            "8" : Bool;
            "9" : Bool;
            "10" : Bool;
            "11" : Bool;
            "12" : Bool;
            "13" : Bool;
            "14" : Bool;
            "15" : Bool;
            "16" : Bool;
         END_STRUCT;
         Spare_4 : Struct
            "1" : Bool;
            "2" : Bool;
            "3" : Bool;
            "4" : Bool;
            "5" : Bool;
            "6" : Bool;
            "7" : Bool;
            "8" : Bool;
            "9" : Bool;
            "10" : Bool;
            "11" : Bool;
            "12" : Bool;
            "13" : Bool;
            "14" : Bool;
            "15" : Bool;
            "16" : Bool;
         END_STRUCT;
      END_STRUCT;
      MES_Error : Struct
         Offline : Bool;   // MES离线
         Reserved1_8 : Bool;
         CheckInCompOverTime_1 : Bool;   // 心跳故障
         CheckInResultOverTime_1 : Bool;
         CheckInCompOverTime_2 : Bool;   // 二维码对比失败
         CheckInResultOverTime_2 : Bool;   // 获取打标数据NG
         CheckInCompOverTime_3 : Bool;   // 获取打标数据超时
         CheckInResultOverTime_3 : Bool;   // 缓存数据和MES数据对比不合格，步序错误 需初始化
         CheckInCompOverTime_4 : Bool;
         CheckInResultOverTime_4 : Bool;   // 主件查询完成超时
         CheckInCompOverTime_5 : Bool;   // 主件查询结果NG
         CheckInResultOverTime_5 : Bool;   // 主件查询完成复位超时
         CheckInCompOverTime_6 : Bool;
         CheckInResultOverTime_6 : Bool;
         CheckInCompOverTime_7 : Bool;
         CheckInResultOverTime_7 : Bool;   // 主件保存完成超时
         CheckInCompOverTime_8 : Bool;   // 主件保存结果反馈超时
         CheckInResultOverTime_8 : Bool;   // 主件保存触发错误
         CheckoutSaveResultNG : Bool;   // 主件保存结果NG
         CheckoutCompRstOverTime : Bool;   // 主件保存完成复位超时
         Reserved2_5 : Bool;
         Reserved2_6 : Bool;
         Reserved2_7 : Bool;
         SubCheck_CompOverTime : Bool;   // 子件查询完成超时
         SubCheck_ResultOverTime : Bool;   // 子件查询结果反馈超时
         SubCheck_TriggerError : Bool;   // 子件查询触发错误
         SubCheck_CheckResultNG : Bool;   // 子件查询结果NG
         SubCheck_CompRstOverTime : Bool;   // 子件查询完成复位超时
         Reserved3_5 : Bool;
         Reserved3_6 : Bool;
         Reserved3_7 : Bool;
         Processing_CompOverTime : Bool;   // 加工不可逆标记完成超时
         Reserved4_1 : Bool;
         Processing_TriggerError : Bool;   // 加工不可逆标记触发错误
         Reserved4_3 : Bool;
         Processing_CompRstOverTime : Bool;   // 加工不可逆标记完成复位超时
         Reserved4_5 : Bool;
         Reserved4_6 : Bool;
         Reserved4_7 : Bool;
         Reserved5_0 : Bool;
         Reserved5_1 : Bool;
         Reserved5_2 : Bool;
         Reserved5_3 : Bool;
         Reserved5_4 : Bool;
         Reserved5_5 : Bool;
         Reserved5_6 : Bool;
         Reserved5_7 : Bool;
      END_STRUCT;
   END_VAR
BEGIN
END_DATA_BLOCK

DATA_BLOCK "ST10_GlobalError"   // DB1066
{ S7_Optimized_Access := 'FALSE' }
// stored: AutoNumber false
   VAR RETAIN
      COM : Struct
         MainPneumaticPressure1NOK : Bool;   // Main Pneumatic pressure 1 NOK,pls check inptut Ix.x,then check if the main valve is opened
         MainPneumaticPressure2NOK : Bool;   // Main Pneumatic pressure 2 NOK,pls check inptut Ix.x,then check if the main valve is opened
         MainPneumaticPressure3NOK : Bool;   // Main Pneumatic pressure 3 NOK,pls check inptut Ix.x,then check if the main valve is opened
         StationNotInHP : Bool;   // Station not in Home position,can't start cycle,pls check the Home positiong state
         CabinetTemperatureNotOk : Bool;   // Cabinet Temperature not OK, please check input Ix.x,then check if the cooling and fan is working
         CoolingUnitNotOk : Bool;   // Cooling unit not OK,pls check input Ix.x,then check if the cooling and fan is working
         RotateTablePositionNOK : Bool;   // The position of the rotate table is not correct after change mode.pls reset position by manual
         RotateTableNotInPosition : Bool;   // No position signal after rotate table Stopped,please check table position and input Ix.x
         StationHardwareError : Bool;
         ChangeStyleError : Bool;
         Reserve3 : Bool;
         Reserve4 : Bool;
         Reserve5 : Bool;
         Reserve6 : Bool;
         Reserve7 : Bool;
         Reserve8 : Bool;
         Reserve : Array[1..4, 0..15] of Bool;
      END_STRUCT;
      Hardware : Struct
         PNSlaveStation01 : Array[1..10] of Struct
            Error : Bool;   // PLC Local Module Error,please check the error module,PLC hardware configuration and online monitor the PLC error message
            Reserve1 : Bool;
            Reserve2 : Bool;
         END_STRUCT;
         COMM : Array[1..5] of Struct   // Communication
            CommunicationError : Bool;   // Serial Communication error,please check power, hardware configuration and connection cable
            NoReceive : Bool;   // Serial Communication receive no information, please check the module settings and communication equipment is the same, check the communication line is the intersection or straight line
            ReceiveWrong : Bool;   // Serial Communication receive the information is wrong, please check the data area is updated in real time
            Reserve1 : Bool;
            Reserve2 : Bool;
         END_STRUCT;
         PNSlaveStation02 : Array[1..10] of Struct   // Substation
            Error : Bool;   // SubStation Missing, please check power, hardware configuration and connection cable
            Reserve1 : Bool;   // SubStation error, please check Slave error code, check the error information in the PLC online hardware
            Reserve2 : Bool;
            Reserve3 : Bool;
         END_STRUCT;
         PNSlaveStation03 : Array[1..10] of Struct   // Remote I/O Error (远程I/O错误）
            Error : Bool;   // Remote I/O communication error, please check the power and communication cable, check the hardware configuration of PLC
            Reserve1 : Bool;   // Remote I/O error, please online monitor the PLC error message
            Reserve2 : Bool;
            Reserve3 : Bool;
         END_STRUCT;
         ValveIsland : Array[1..5] of Struct   // Valve Island Error（阀岛错误）
            SystemError : Bool;   // Valve island error, pls check the error code , check the error information in the PLC online hardware
            OffLine : Bool;   // Valve island is lost, pls check the island's cable , check valve island in PLC configuration and the actual agreement
            Reserve1 : Bool;
            Reserve2 : Bool;
         END_STRUCT;
      END_STRUCT;
      Safety : Struct
         "Robot 1 Estop" : Bool;   // Safety circuit not OK,pls check input Ix.x,then check if the safety circuit control on
         "Robot 2 Estop" : Bool;   // E-stop safety circuit not OK, please check input Ix.x, then reset safety circurt
         HMIEstopPBActivated : Bool;   // HMI Estop PB Activated，pls check input Ix.x,then check Estop button,if Estop button is close,pls open the Estop button
         TableEstopPB1Activated : Bool;   // HTable Estop PB1 Activated，pls check input Ix.x,then check Estop button,if Estop button is close,pls open the Estop button
         TableEstopPB2Activated : Bool;   // Table Estop PB2 Activated，pls check input Ix.x,then check Estop button,if Estop button is close,pls open the Estop button
         TableEstopPB3Activated : Bool;   // Table Estop PB3 Activated，pls check input Ix.x,then check Estop button,if Estop button is close,pls open the Estop button
         TableEstopPB4Activated : Bool;   // Table Estop PB4 Activated，pls check input Ix.x,then check Estop button,if Estop button is close,pls open the Estop button
         TableEstopPB5Activated : Bool;   // Table Estop PB5 Activated，pls check input Ix.x,then check Estop button,if Estop button is close,pls open the Estop button
         TableEstopPB6Activated : Bool;   // Table Estop PB6 Activated，pls check input Ix.x,then check Estop button,if Estop button is close,pls open the Estop button
         EStopSafety : Bool;
         TableEstopPB7Activated : Bool;
         TableEstopPB8Activated : Bool;
         TableEstopPB9Activated : Bool;
         StoveEstopActivated : Bool;
         "Robot 3 Estop" : Bool;
         Reserve9 : Bool;
         Reserve : Array[1..4, 0..15] of Bool;
      END_STRUCT;
      SafetyDoor : Struct
         "Type" : Array[1..5] of Struct   // Safety Door circuit type
            NotOk : Bool;   // Safety Door type [*] circuit not OK, please check input Ix.x, then reset safety circurt
            OpenInRunning : Bool;   // The safety door is opened when device Running,pls power on than initialize device
            Reserve1 : Bool;
            Reserve2 : Bool;
         END_STRUCT;
         No : Array[1..9] of Struct   // SafetyDoorNumber
            NotLock : Bool;   // Safety door lock is not lock，pls check input Ix.x，then check safety door lock output Qx.x
            Notlocked : Bool;   // Safety door lock is not unlock，pls check input Ix.x，then check safety door lock output Qx.x
            NotClose : Bool;   // Safety door is not close,pls check satety door lock position
            Reserve1 : Bool;
            Reserve2 : Bool;
         END_STRUCT;
         MaterialDoor : Struct
            NotLock_1 : Bool;
            NotClose_1 : Bool;
            NotLock_2 : Bool;
            NotClose_2 : Bool;
            NotLock_3 : Bool;
            NotClose_3 : Bool;
            NotLock_4 : Bool;
            NotClose_4 : Bool;
            NotLock_5 : Bool;
            NotClose_5 : Bool;
            NotLock_6 : Bool;
            NotClose_6 : Bool;
            NotLock_7 : Bool;
            NotClose_7 : Bool;
            NotLock_8 : Bool;
            NotClose_8 : Bool;
         END_STRUCT;
      END_STRUCT;
      LightCurtain : Array[1..5] of Struct
         ActivatedInRunning : Bool;   // Light curtain is Activated when device Running, pls power on than initialize device
         ActivatedInRotTableRun : Bool;   // Light curtain is Activated when rotate table running,please press the reset button to rotate the rotate table to position
         Error : Bool;   // Light curtain error,pls check the light curtain connection or check the error code
         Reserve1 : Bool;
         Reserve2 : Bool;
      END_STRUCT;
      Product : Array[1..5] of Struct
         TypeSelectionError : Bool;   // Product Type selection error,pls select the proper type
         TypeWrong : Bool;   // Product is not match current model, please make sure the product model is entered correctly
         NotforStation : Bool;   // Product not for this station,pls check if the Product is proper
         TypeAutoChangeError : Bool;
         Reserve2 : Bool;
      END_STRUCT;
      Fixture : Array[1..10] of Struct
         PositionError : Bool;   // Fixture [*] position error,pls put the fixture on proper positon
         TypeError : Bool;   // Fixture [*] tpye error,pls put the correct fixture into the tooling
         Reserve1 : Bool;
         Reserve2 : Bool;
      END_STRUCT;
      Breaker : Struct   // Power Breaker
         Trip : Array[1..16] of Bool;   // Breaker tripped, please check input Ix.x
      END_STRUCT;
   END_VAR
BEGIN
END_DATA_BLOCK

DATA_BLOCK "ST10_WarningDB"   // DB1068
{ S7_Optimized_Access := 'FALSE' }
// stored: AutoNumber false
   VAR RETAIN
      Global : Struct   // Global Warning（通用警告）
         "1" : Struct
            PartLack1 : Bool;   // The main part1 lack
            PartLack2 : Bool;   // The part2 lack
            PartLack3 : Bool;   // The part3 lack
            PartLack4 : Bool;   // The part4 lack
            PartLack5 : Bool;   // The part5 lack
            PartLack6 : Bool;   // The part6 lack
            PartLack7 : Bool;   // The part7 lack
            PartLack8 : Bool;   // The part8 lack
         END_STRUCT;
         "2" : Array[0..15] of Bool;
         "3" : Struct
            PartNoProperPosition1 : Bool;   // The main part1 no proper position
            PartNoProperPosition2 : Bool;   // The part2 no proper position
            PartNoProperPosition3 : Bool;   // The part3 no proper position
            PartNoProperPosition4 : Bool;   // The part4 no proper position
            PartNoProperPosition5 : Bool;   // The part5 no proper position
            PartNoProperPosition6 : Bool;   // The part6 no proper position
            PartNoProperPosition7 : Bool;   // The part7 no proper position
            PartNoProperPosition8 : Bool;   // The part8 no proper position
         END_STRUCT;
         "4" : Array[0..15] of Bool;
         "5" : Struct
            ChangoverDataInvalide : Bool;   // The changover data invalide
            PartDateInvalide : Bool;   // The part date invalide
            StationInHPToStart : Bool;   // The station has to be at base pos to start
            lastStationPartNok : Bool;   // The last station part is Nok
         END_STRUCT;
         "6" : Array[0..15] of Bool;
         "7" : Array[0..15] of Bool;
         "8" : Array[0..15] of Bool;
         "9" : Array[0..15] of Bool;
         "10" : Array[0..15] of Bool;
      END_STRUCT;
      IndexTable : Array[1..2, 0..15] of Bool;   // Indextable Warning（转台警告）
      Serve : Array[1..2, 0..15] of Bool;   // Serve Warning（伺服警告）
      Servepress : Array[1..2, 0..15] of Bool;   // Serve press Warning（伺服压机警告）
      "3AxisServoInterpolation" : Array[1..2, 0..15] of Bool;   // Servo Motor Risk Money(3 axis)Warning （伺服电机3轴差补系统警告）
      LaserWelding : Array[1..2, 0..15] of Bool;   // Laser Welding Warning(激光焊接机警告)
      LaserMarking : Array[1..2, 0..15] of Bool;   // Laser Marking Warning(激光打标机警告)
      Printer : Array[1..2, 0..15] of Bool;   // Printer Warning(打印机警告)
      Marking : Array[1..2, 0..15] of Bool;   // Marking Warning(标识机警告)
      Labelling : Array[1..2, 0..15] of Bool;   // Labelling Warning（贴标机警告）
      Dispensing : Array[1..2, 0..15] of Bool;   // Dispensing Warning（点胶警告）
      GreasingSystem : Array[1..2, 0..15] of Bool;   // Greasing System Warning(注油系统警告）
      HotWindSystem : Array[1..2, 0..15] of Bool;   // Hot Wind System Warning(热风系统警告）
      HighFrequencyHeating : Array[1..2, 0..15] of Bool;   // High Frequency Heating Warning（高频加热警告）
      Degaussing : Array[1..2, 0..15] of Bool;   // Degaussing Warning（消磁警告）
      BowlFeeder : Array[1..2, 0..15] of Bool;   // Bowl Feeder Warning（振动盘警告）
      Riveter : Array[1..2, 0..15] of Bool;   // Riveter Warning（铆接机警告）
      HydraulicSystem : Array[1..2, 0..15] of Bool;   // Hydraulic System Warning（液压系统警告）
      Robot : Array[1..2, 0..15] of Bool;   // Robot Warning（机器人警告）
      Camera : Array[1..2, 0..15] of Bool;   // Camera Warning(影像警告)
      Scannner : Array[1..2, 0..15] of Bool;   // Scannner Warning(读码警告)
      MeasureSensor : Array[1..2, 0..15] of Bool;   // Measure Sensor Warning(测量传感器警告)
      Leakage : Array[1..2, 0..15] of Bool;   // Leakage Warning（泄露测试仪警告）
      TestPowerSupply : Array[1..2, 0..15] of Bool;   // Test Power Supply Warning (测试电源警告）
      HighVoltageTester : Array[1..2, 0..15] of Bool;   // High Voltage Test Warning(高压测试警告）
      EOLfinalInspection : Array[1..2, 0..15] of Bool;   // EOL final inspection Warning（EOL终检测试警告）
      Screw : Array[1..2, 0..15] of Bool;   // Screw Warning(电动螺丝刀警告)
      "3AxisScrewEncoder" : Array[1..2, 0..15] of Bool;   // Screw Encoder(3 axis)Warning(螺丝刀编码器警告）
      Heating : Array[1..2, 0..15] of Bool;   // Heating Warning（加热警告）
      PressurizedOilAirCylinder : Array[1..2, 0..15] of Bool;   // Pressurized Oil-Air Cylinder Warning(气液增力缸警告）
      Moby : Array[1..2, 0..15] of Bool;   // Moby Warning(Moby警告)
      IPC : Array[1..2, 0..15] of Bool;   // IPC Warning（服务器警告）
      ValveIsland : Array[1..2, 0..15] of Bool;   // Valve island Warning (阀岛警告）
      RFID : Array[1..2, 0..15] of Bool;   // RFID Warning（无线射频识别警告）
      RemoteIO : Array[1..2, 0..15] of Bool;   // Remote I/O Warning（远程I/O警告）
      DPSlaveStation : Array[1..2, 0..15] of Bool;   // DP Slave Station Warning（DP从站警告）
      MSCOMM : Array[1..2, 0..15] of Bool;   // MSCOMM Warning（串口通讯警告）
      Flowtester : Array[1..2, 0..15] of Bool;   // Flow tester Warning（流量测试仪错误）
      CurrentsTester : Array[1..2, 0..15] of Bool;   // Currents Tester Warning(电流测试仪)）
      VoltageTester : Array[1..2, 0..15] of Bool;   // Voltage Tester Warning(电压测试仪)
      InductanceTester : Array[1..2, 0..15] of Bool;   // Inductance Tester Warning(电感测试仪)
      ResistanceTester : Array[1..2, 0..15] of Bool;   // Resistance Tester Warning(电阻测试仪)
      LCRTester : Array[1..2, 0..15] of Bool;   // LCR Test Warning(LCR测试)
      PressureDisplacementMonitor : Array[1..2, 0..15] of Bool;   // Pressure Displacement Monitor Warning(压力位移监控仪)
      UltrasonicWelding : Array[1..2, 0..15] of Bool;   // Ultrasonic Welding Warning(超声波焊接)
      ElectricResistanceWelding : Array[1..2, 0..15] of Bool;   // Electric Resistance Welding Warning(电阻焊)
   END_VAR
BEGIN
END_DATA_BLOCK

DATA_BLOCK "ST10_TipDB"   // DB1069
{ S7_Optimized_Access := 'FALSE' }
// stored: AutoNumber false
   VAR RETAIN
      Global : Struct
         "1" : Struct
            ControlOn : Bool;   // 7000:提示：设备未上电，请先按复位按钮，再按控制开按钮
            closesafetyDoor : Bool;   // 7001:提示：设备存在故障，请查看报警信息，消除故障，然后按复位按钮
            LockSafetyDoor : Bool;   // 7003:提示：设备未选择自动，请选择自动模式
            SelectAutoMode : Bool;   // 7005:提示：设备未启动，请启动自动运行
            SelectManualMode : Bool;
            AutoModeRunning : Bool;
            SafetyDoorLocked : Bool;
            SaferyDoorNotLocked : Bool;
            GoWP : Bool;
            Reset : Bool;
         END_STRUCT;
         "2" : Array[0..15] of Bool;
         "3" : Array[0..15] of Bool;
         "4" : Array[0..15] of Bool;
         "5" : Struct
            FuncrionDeactive1 : Bool;
            FuncrionDeactive2 : Bool;
            FuncrionDeactive3 : Bool;
            FuncrionDeactive4 : Bool;
            FuncrionDeactive5 : Bool;
            FuncrionDeactive6 : Bool;
            FuncrionDeactive7 : Bool;
            FuncrionDeactive8 : Bool;
         END_STRUCT;
         "6" : Array[0..15] of Bool;
         "7" : Struct
            ScanMainPartDMC1 : Bool;
            ScanPartDMC2 : Bool;
            ScanPartDMC3 : Bool;
            ScanPartDMC4 : Bool;
            ScanPartDMC5 : Bool;
            ScanPartDMC6 : Bool;
            ScanPartDMC7 : Bool;
            ScanPartDMC8 : Bool;
         END_STRUCT;
         "8" : Array[0..15] of Bool;
         "9" : Array[0..15] of Bool;
         "10" : Array[0..15] of Bool;
      END_STRUCT;
      OP1 : Struct   // ST70_B_提示信息
         "Take off product" : Bool;   // 请取下托盘上产品
         "Put product" : Bool;   // 请放入转向器壳体总成
         "Please scan the code" : Bool;   // 请扫转向器壳体总成二维码
         "Please apply Oil" : Bool;   // 请手持涂油工装涂油
         "Please take the O-ring" : Bool;   // 请取O型圈并安装完成
         "Please put in the powertrain" : Bool;   // 请扫转向器总成二维码
         Static_2 : Bool;
         "Please pre-screw" : Bool;   // 请安装转向器动力总成并预拧螺丝
         Static_1 : Bool;
         Static_3 : Bool;
         "Please press the button_1" : Bool;   // 请按下ST70-B启动按钮
         Reset : Bool;   // RFID状态数据未清除，请复位清除数据
      END_STRUCT;
      OP2 : Struct   // ST70_C_提示信息
         Static_4 : Bool;
         Static_2 : Bool;
         Static_3 : Bool;
         "Please press the button" : Bool;   // 请按下ST70_C启动按钮
         "Please press the trigger" : Bool;   // 请按下螺丝枪扳机拧紧螺丝
         "Please take the paint pen" : Bool;   // 请取出油漆笔划上标识
         "Please put back the paint pen" : Bool;   // 请划上标识后放回油漆笔
         Static_1 : Bool;
         "Please remove the product" : Bool;   // 产品报废,请取下产品
         "Please press the screw gun trigger" : Bool;   // 重新拧紧,请按下螺丝枪扳机
      END_STRUCT;
   END_VAR
BEGIN
   // Global."2"[0] : 7002:提示：未选择配方，请在换型页面选择配方
   // Global."2"[1] : 7004:提示：设备未初始化，请启动初始化
END_DATA_BLOCK

DATA_BLOCK "Parameter"   // DB170
{ S7_Optimized_Access := 'TRUE' }
// stored: AutoNumber false, IsRetainMemResEnabled true, MemoryReserve 10000
   VAR RETAIN
      AxisRun : Struct
         Axis : Array[1..15] of "ServoType_UDT";
      END_STRUCT;
      AxisNuw : Struct
         Axis : Array[1..15] of "ServoType_UDT";
      END_STRUCT;
      AxisDisplay : Struct
         Axis : Array[1..15] of "ServoType_UDT";
      END_STRUCT;
      AxisSave : Struct
         Axis : Array[1..15] of "ServoType_UDT";
      END_STRUCT;
      AxisStore : Array[1..15] of Struct
         Axis : Array[1..15] of "ServoType_UDT";
      END_STRUCT;
   END_VAR
BEGIN
   // AxisRun.Axis[1].Pos1 : 上料位1
   // AxisRun.Axis[2].Pos1 : 初始位
   // AxisRun.Axis[3].Pos1 : 初始位/IV拍照位_1
   // AxisRun.Axis[4].Pos1 : 上料位1
   // AxisRun.Axis[5].Pos1 : Z轴初始位
   // AxisRun.Axis[6].Pos1 : X轴初始位
   // AxisRun.Axis[7].Pos1 : Y轴初始位
   AxisRun.Axis[1].Pos1.Position := 3.419;
   AxisRun.Axis[2..3].Pos1.Position := 0.0;
   AxisRun.Axis[4].Pos1.Position := 3.585;
   AxisRun.Axis[5].Pos1.Position := 143.76;
   AxisRun.Axis[6].Pos1.Position := 2.34;
   AxisRun.Axis[7].Pos1.Position := 115.47;
   AxisRun.Axis[8..15].Pos1.Position := 0.0;
   AxisRun.Axis[1..2].Pos1.Speed := 10000;
   AxisRun.Axis[3].Pos1.Speed := 20000;
   AxisRun.Axis[4].Pos1.Speed := 10000;
   AxisRun.Axis[5..7].Pos1.Speed := 200;
   AxisRun.Axis[8..15].Pos1.Speed := 0;
   AxisRun.Axis[1..15].Pos1.Reached := FALSE;
   // AxisRun.Axis[1].Pos2 : 上料位2
   // AxisRun.Axis[2].Pos2 : 扫码位置2
   // AxisRun.Axis[3].Pos2 : 点胶1结束位
   // AxisRun.Axis[4].Pos2 : 上料位2
   // AxisRun.Axis[5].Pos2 : Z轴点胶位1
   // AxisRun.Axis[6].Pos2 : X轴点胶等待位
   // AxisRun.Axis[7].Pos2 : Y轴点胶位1
   AxisRun.Axis[1].Pos2.Position := 48.386;
   AxisRun.Axis[2].Pos2.Position := 450.0;
   AxisRun.Axis[3].Pos2.Position := 490.0;
   AxisRun.Axis[4].Pos2.Position := 48.61;
   AxisRun.Axis[5].Pos2.Position := 143.76;
   AxisRun.Axis[6].Pos2.Position := 76.0;
   AxisRun.Axis[7].Pos2.Position := 115.47;
   AxisRun.Axis[8..15].Pos2.Position := 0.0;
   AxisRun.Axis[1..4].Pos2.Speed := 10000;
   AxisRun.Axis[5..7].Pos2.Speed := 200;
   AxisRun.Axis[8..15].Pos2.Speed := 0;
   AxisRun.Axis[1..15].Pos2.Reached := FALSE;
   // AxisRun.Axis[1].Pos3 : 上料位3
   // AxisRun.Axis[2].Pos3 : 扫码位置3
   // AxisRun.Axis[3].Pos3 : 点胶2结束位
   // AxisRun.Axis[4].Pos3 : 上料位3
   // AxisRun.Axis[5].Pos3 : Z轴点胶位2
   // AxisRun.Axis[6].Pos3 : X轴点胶位1
   // AxisRun.Axis[7].Pos3 : Y轴点胶位2
   AxisRun.Axis[1].Pos3.Position := 93.294;
   AxisRun.Axis[2].Pos3.Position := 900.0;
   AxisRun.Axis[3].Pos3.Position := 490.0;
   AxisRun.Axis[4].Pos3.Position := 93.637;
   AxisRun.Axis[5].Pos3.Position := 137.76;
   AxisRun.Axis[6].Pos3.Position := 84.69;
   AxisRun.Axis[7].Pos3.Position := 115.47;
   AxisRun.Axis[8..15].Pos3.Position := 0.0;
   AxisRun.Axis[1..4].Pos3.Speed := 10000;
   AxisRun.Axis[5..7].Pos3.Speed := 200;
   AxisRun.Axis[8..15].Pos3.Speed := 0;
   AxisRun.Axis[1..15].Pos3.Reached := FALSE;
   // AxisRun.Axis[1].Pos4 : 上料位4
   // AxisRun.Axis[2].Pos4 : 扫码位置4
   // AxisRun.Axis[3].Pos4 : 点胶3结束位
   // AxisRun.Axis[4].Pos4 : 上料位4
   // AxisRun.Axis[5].Pos4 : Z轴点胶位3
   // AxisRun.Axis[6].Pos4 : X轴点胶位2
   // AxisRun.Axis[7].Pos4 : Y轴点胶位3
   AxisRun.Axis[1].Pos4.Position := 138.335;
   AxisRun.Axis[2].Pos4.Position := 135.0;
   AxisRun.Axis[3].Pos4.Position := 490.0;
   AxisRun.Axis[4].Pos4.Position := 138.606;
   AxisRun.Axis[5].Pos4.Position := 130.36;
   AxisRun.Axis[6].Pos4.Position := 84.69;
   AxisRun.Axis[7].Pos4.Position := 115.47;
   AxisRun.Axis[8..15].Pos4.Position := 0.0;
   AxisRun.Axis[1..4].Pos4.Speed := 10000;
   AxisRun.Axis[5..7].Pos4.Speed := 200;
   AxisRun.Axis[8..15].Pos4.Speed := 0;
   AxisRun.Axis[1..15].Pos4.Reached := FALSE;
   // AxisRun.Axis[1].Pos5 : 上料位5
   // AxisRun.Axis[2].Pos5 : 扫码位置5
   // AxisRun.Axis[3].Pos5 : 点胶4结束位//点胶位置取消
   // AxisRun.Axis[4].Pos5 : 上料位5
   // AxisRun.Axis[5].Pos5 : Z轴点胶位4
   // AxisRun.Axis[6].Pos5 : X轴点胶位3
   // AxisRun.Axis[7].Pos5 : Y轴点胶位4
   AxisRun.Axis[1].Pos5.Position := 183.464;
   AxisRun.Axis[2].Pos5.Position := 180.0;
   AxisRun.Axis[3].Pos5.Position := 0.0;
   AxisRun.Axis[4].Pos5.Position := 183.388;
   AxisRun.Axis[5].Pos5.Position := 124.16;
   AxisRun.Axis[6].Pos5.Position := 84.69;
   AxisRun.Axis[7].Pos5.Position := 115.47;
   AxisRun.Axis[8..15].Pos5.Position := 0.0;
   AxisRun.Axis[1..2].Pos5.Speed := 10000;
   AxisRun.Axis[3].Pos5.Speed := 0;
   AxisRun.Axis[4].Pos5.Speed := 10000;
   AxisRun.Axis[5..7].Pos5.Speed := 200;
   AxisRun.Axis[8..15].Pos5.Speed := 0;
   AxisRun.Axis[1..15].Pos5.Reached := FALSE;
   // AxisRun.Axis[1].Pos6 : 上料位6
   // AxisRun.Axis[2].Pos6 : 扫码位置6
   // AxisRun.Axis[3].Pos6 : 点胶5结束位
   // AxisRun.Axis[4].Pos6 : 上料位6
   // AxisRun.Axis[5].Pos6 : Z轴点胶位5
   // AxisRun.Axis[6].Pos6 : X轴点胶位4
   // AxisRun.Axis[7].Pos6 : Y轴点胶位5
   AxisRun.Axis[1].Pos6.Position := 228.443;
   AxisRun.Axis[2].Pos6.Position := 225.0;
   AxisRun.Axis[3].Pos6.Position := 490.0;
   AxisRun.Axis[4].Pos6.Position := 228.458;
   AxisRun.Axis[5].Pos6.Position := 125.65;
   AxisRun.Axis[6].Pos6.Position := 84.69;
   AxisRun.Axis[7].Pos6.Position := 110.18;
   AxisRun.Axis[8..15].Pos6.Position := 0.0;
   AxisRun.Axis[1..4].Pos6.Speed := 10000;
   AxisRun.Axis[5..7].Pos6.Speed := 200;
   AxisRun.Axis[8..15].Pos6.Speed := 0;
   AxisRun.Axis[1..15].Pos6.Reached := FALSE;
   // AxisRun.Axis[1].Pos7 : 上料位7
   // AxisRun.Axis[2].Pos7 : 扫码位置7
   // AxisRun.Axis[3].Pos7 : IV拍照位_2
   // AxisRun.Axis[4].Pos7 : 上料位7
   // AxisRun.Axis[5].Pos7 : Z轴相机检测位
   // AxisRun.Axis[6].Pos7 : X轴点胶位5
   // AxisRun.Axis[7].Pos7 : Y轴相机检测位
   AxisRun.Axis[1].Pos7.Position := 273.535;
   AxisRun.Axis[2].Pos7.Position := 270.0;
   AxisRun.Axis[3].Pos7.Position := 90.0;
   AxisRun.Axis[4].Pos7.Position := 273.513;
   AxisRun.Axis[5].Pos7.Position := 48.11;
   AxisRun.Axis[6].Pos7.Position := 85.0;
   AxisRun.Axis[7].Pos7.Position := 60.52;
   AxisRun.Axis[8..15].Pos7.Position := 0.0;
   AxisRun.Axis[1..4].Pos7.Speed := 10000;
   AxisRun.Axis[5..7].Pos7.Speed := 200;
   AxisRun.Axis[8..15].Pos7.Speed := 0;
   AxisRun.Axis[1..15].Pos7.Reached := FALSE;
   // AxisRun.Axis[1].Pos8 : 上料位8
   // AxisRun.Axis[2].Pos8 : 扫码位置8
   // AxisRun.Axis[3].Pos8 : IV拍照位_3
   // AxisRun.Axis[4].Pos8 : 上料位8
   // AxisRun.Axis[5].Pos8 : Z轴原点位
   // AxisRun.Axis[6].Pos8 : X轴相机检测位
   AxisRun.Axis[1].Pos8.Position := 318.25;
   AxisRun.Axis[2].Pos8.Position := 315.0;
   AxisRun.Axis[3].Pos8.Position := 180.0;
   AxisRun.Axis[4].Pos8.Position := 318.501;
   AxisRun.Axis[5].Pos8.Position := 0.0;
   AxisRun.Axis[6].Pos8.Position := 88.53;
   AxisRun.Axis[7].Pos8.Position := 80.0;
   AxisRun.Axis[8..15].Pos8.Position := 0.0;
   AxisRun.Axis[1..4].Pos8.Speed := 10000;
   AxisRun.Axis[5..6].Pos8.Speed := 200;
   AxisRun.Axis[7].Pos8.Speed := 100;
   AxisRun.Axis[8..15].Pos8.Speed := 0;
   AxisRun.Axis[1..15].Pos8.Reached := FALSE;
   // AxisRun.Axis[3].Pos9 : IV拍照位_4
   // AxisRun.Axis[5].Pos9 : Z轴Up点胶位5
   AxisRun.Axis[1..2].Pos9.Position := 0.0;
   AxisRun.Axis[3].Pos9.Position := 270.0;
   AxisRun.Axis[4].Pos9.Position := 0.0;
   AxisRun.Axis[5].Pos9.Position := 48.11;
   AxisRun.Axis[6..15].Pos9.Position := 0.0;
   AxisRun.Axis[1..2].Pos9.Speed := 0;
   AxisRun.Axis[3].Pos9.Speed := 10000;
   AxisRun.Axis[4].Pos9.Speed := 0;
   AxisRun.Axis[5].Pos9.Speed := 200;
   AxisRun.Axis[6..15].Pos9.Speed := 0;
   AxisRun.Axis[1..15].Pos9.Reached := FALSE;
   AxisRun.Axis[1..15].Pos10.Position := 0.0;
   AxisRun.Axis[1..15].Pos10.Speed := 0;
   AxisRun.Axis[1..15].Pos10.Reached := FALSE;
   AxisRun.Axis[1..15].Pos11.Position := 0.0;
   AxisRun.Axis[1..15].Pos11.Speed := 0;
   AxisRun.Axis[1..15].Pos11.Reached := FALSE;
   AxisRun.Axis[1..15].Pos12.Position := 0.0;
   AxisRun.Axis[1..15].Pos12.Speed := 0;
   AxisRun.Axis[1..15].Pos12.Reached := FALSE;
   AxisRun.Axis[1..15].Pos13.Position := 0.0;
   AxisRun.Axis[1..15].Pos13.Speed := 0;
   AxisRun.Axis[1..15].Pos13.Reached := FALSE;
   AxisRun.Axis[1..15].Pos14.Position := 0.0;
   AxisRun.Axis[1..15].Pos14.Speed := 0;
   AxisRun.Axis[1..15].Pos14.Reached := FALSE;
   AxisRun.Axis[1..15].Pos15.Position := 0.0;
   AxisRun.Axis[1..15].Pos15.Speed := 0;
   AxisRun.Axis[1..15].Pos15.Reached := FALSE;
   AxisRun.Axis[1..15].Pos16.Position := 0.0;
   AxisRun.Axis[1..15].Pos16.Speed := 0;
   AxisRun.Axis[1..15].Pos16.Reached := FALSE;
   AxisRun.Axis[1..15].Pos17.Position := 0.0;
   AxisRun.Axis[1..15].Pos17.Speed := 0;
   AxisRun.Axis[1..15].Pos17.Reached := FALSE;
   AxisRun.Axis[1..15].Pos18.Position := 0.0;
   AxisRun.Axis[1..15].Pos18.Speed := 0;
   AxisRun.Axis[1..15].Pos18.Reached := FALSE;
   AxisRun.Axis[1..15].Pos19.Position := 0.0;
   AxisRun.Axis[1..15].Pos19.Speed := 0;
   AxisRun.Axis[1..15].Pos19.Reached := FALSE;
   AxisRun.Axis[1..15].Pos20.Position := 0.0;
   AxisRun.Axis[1..15].Pos20.Speed := 0;
   AxisRun.Axis[1..15].Pos20.Reached := FALSE;
   AxisRun.Axis[1..15].Pos21.Position := 0.0;
   AxisRun.Axis[1..15].Pos21.Speed := 0;
   AxisRun.Axis[1..15].Pos21.Reached := FALSE;
   AxisRun.Axis[1..15].Pos22.Position := 0.0;
   AxisRun.Axis[1..15].Pos22.Speed := 0;
   AxisRun.Axis[1..15].Pos22.Reached := FALSE;
   AxisRun.Axis[1..15].Pos23.Position := 0.0;
   AxisRun.Axis[1..15].Pos23.Speed := 0;
   AxisRun.Axis[1..15].Pos23.Reached := FALSE;
   AxisRun.Axis[1..15].Pos24.Position := 0.0;
   AxisRun.Axis[1..15].Pos24.Speed := 0;
   AxisRun.Axis[1..15].Pos24.Reached := FALSE;
   AxisRun.Axis[1..15].Pos25.Position := 0.0;
   AxisRun.Axis[1..15].Pos25.Speed := 0;
   AxisRun.Axis[1..15].Pos25.Reached := FALSE;
   AxisRun.Axis[1..15].Pos26.Position := 0.0;
   AxisRun.Axis[1..15].Pos26.Speed := 0;
   AxisRun.Axis[1..15].Pos26.Reached := FALSE;
   AxisRun.Axis[1..15].Pos27.Position := 0.0;
   AxisRun.Axis[1..15].Pos27.Speed := 0;
   AxisRun.Axis[1..15].Pos27.Reached := FALSE;
   AxisRun.Axis[1..15].Pos28.Position := 0.0;
   AxisRun.Axis[1..15].Pos28.Speed := 0;
   AxisRun.Axis[1..15].Pos28.Reached := FALSE;
   AxisRun.Axis[1..15].Pos29.Position := 0.0;
   AxisRun.Axis[1..15].Pos29.Speed := 0;
   AxisRun.Axis[1..15].Pos29.Reached := FALSE;
   AxisRun.Axis[1..15].Pos30.Position := 0.0;
   AxisRun.Axis[1..15].Pos30.Speed := 0;
   AxisRun.Axis[1..15].Pos30.Reached := FALSE;
   AxisNuw.Axis[1..15].Pos1.Position := 0.0;
   AxisNuw.Axis[1..15].Pos1.Speed := 0;
   AxisNuw.Axis[1..15].Pos1.Reached := FALSE;
   AxisNuw.Axis[1..15].Pos2.Position := 0.0;
   AxisNuw.Axis[1..15].Pos2.Speed := 0;
   AxisNuw.Axis[1..15].Pos2.Reached := FALSE;
   AxisNuw.Axis[1..15].Pos3.Position := 0.0;
   AxisNuw.Axis[1..15].Pos3.Speed := 0;
   AxisNuw.Axis[1..15].Pos3.Reached := FALSE;
   AxisNuw.Axis[1..15].Pos4.Position := 0.0;
   AxisNuw.Axis[1..15].Pos4.Speed := 0;
   AxisNuw.Axis[1..15].Pos4.Reached := FALSE;
   AxisNuw.Axis[1..15].Pos5.Position := 0.0;
   AxisNuw.Axis[1..15].Pos5.Speed := 0;
   AxisNuw.Axis[1..15].Pos5.Reached := FALSE;
   AxisNuw.Axis[1..15].Pos6.Position := 0.0;
   AxisNuw.Axis[1..15].Pos6.Speed := 0;
   AxisNuw.Axis[1..15].Pos6.Reached := FALSE;
   AxisNuw.Axis[1..15].Pos7.Position := 0.0;
   AxisNuw.Axis[1..15].Pos7.Speed := 0;
   AxisNuw.Axis[1..15].Pos7.Reached := FALSE;
   AxisNuw.Axis[1..15].Pos8.Position := 0.0;
   AxisNuw.Axis[1..15].Pos8.Speed := 0;
   AxisNuw.Axis[1..15].Pos8.Reached := FALSE;
   AxisNuw.Axis[1..15].Pos9.Position := 0.0;
   AxisNuw.Axis[1..15].Pos9.Speed := 0;
   AxisNuw.Axis[1..15].Pos9.Reached := FALSE;
   AxisNuw.Axis[1..15].Pos10.Position := 0.0;
   AxisNuw.Axis[1..15].Pos10.Speed := 0;
   AxisNuw.Axis[1..15].Pos10.Reached := FALSE;
   AxisNuw.Axis[1..15].Pos11.Position := 0.0;
   AxisNuw.Axis[1..15].Pos11.Speed := 0;
   AxisNuw.Axis[1..15].Pos11.Reached := FALSE;
   AxisNuw.Axis[1..15].Pos12.Position := 0.0;
   AxisNuw.Axis[1..15].Pos12.Speed := 0;
   AxisNuw.Axis[1..15].Pos12.Reached := FALSE;
   AxisNuw.Axis[1..15].Pos13.Position := 0.0;
   AxisNuw.Axis[1..15].Pos13.Speed := 0;
   AxisNuw.Axis[1..15].Pos13.Reached := FALSE;
   AxisNuw.Axis[1..15].Pos14.Position := 0.0;
   AxisNuw.Axis[1..15].Pos14.Speed := 0;
   AxisNuw.Axis[1..15].Pos14.Reached := FALSE;
   AxisNuw.Axis[1..15].Pos15.Position := 0.0;
   AxisNuw.Axis[1..15].Pos15.Speed := 0;
   AxisNuw.Axis[1..15].Pos15.Reached := FALSE;
   AxisNuw.Axis[1..15].Pos16.Position := 0.0;
   AxisNuw.Axis[1..15].Pos16.Speed := 0;
   AxisNuw.Axis[1..15].Pos16.Reached := FALSE;
   AxisNuw.Axis[1..15].Pos17.Position := 0.0;
   AxisNuw.Axis[1..15].Pos17.Speed := 0;
   AxisNuw.Axis[1..15].Pos17.Reached := FALSE;
   AxisNuw.Axis[1..15].Pos18.Position := 0.0;
   AxisNuw.Axis[1..15].Pos18.Speed := 0;
   AxisNuw.Axis[1..15].Pos18.Reached := FALSE;
   AxisNuw.Axis[1..15].Pos19.Position := 0.0;
   AxisNuw.Axis[1..15].Pos19.Speed := 0;
   AxisNuw.Axis[1..15].Pos19.Reached := FALSE;
   AxisNuw.Axis[1..15].Pos20.Position := 0.0;
   AxisNuw.Axis[1..15].Pos20.Speed := 0;
   AxisNuw.Axis[1..15].Pos20.Reached := FALSE;
   AxisNuw.Axis[1..15].Pos21.Position := 0.0;
   AxisNuw.Axis[1..15].Pos21.Speed := 0;
   AxisNuw.Axis[1..15].Pos21.Reached := FALSE;
   AxisNuw.Axis[1..15].Pos22.Position := 0.0;
   AxisNuw.Axis[1..15].Pos22.Speed := 0;
   AxisNuw.Axis[1..15].Pos22.Reached := FALSE;
   AxisNuw.Axis[1..15].Pos23.Position := 0.0;
   AxisNuw.Axis[1..15].Pos23.Speed := 0;
   AxisNuw.Axis[1..15].Pos23.Reached := FALSE;
   AxisNuw.Axis[1..15].Pos24.Position := 0.0;
   AxisNuw.Axis[1..15].Pos24.Speed := 0;
   AxisNuw.Axis[1..15].Pos24.Reached := FALSE;
   AxisNuw.Axis[1..15].Pos25.Position := 0.0;
   AxisNuw.Axis[1..15].Pos25.Speed := 0;
   AxisNuw.Axis[1..15].Pos25.Reached := FALSE;
   AxisNuw.Axis[1..15].Pos26.Position := 0.0;
   AxisNuw.Axis[1..15].Pos26.Speed := 0;
   AxisNuw.Axis[1..15].Pos26.Reached := FALSE;
   AxisNuw.Axis[1..15].Pos27.Position := 0.0;
   AxisNuw.Axis[1..15].Pos27.Speed := 0;
   AxisNuw.Axis[1..15].Pos27.Reached := FALSE;
   AxisNuw.Axis[1..15].Pos28.Position := 0.0;
   AxisNuw.Axis[1..15].Pos28.Speed := 0;
   AxisNuw.Axis[1..15].Pos28.Reached := FALSE;
   AxisNuw.Axis[1..15].Pos29.Position := 0.0;
   AxisNuw.Axis[1..15].Pos29.Speed := 0;
   AxisNuw.Axis[1..15].Pos29.Reached := FALSE;
   AxisNuw.Axis[1..15].Pos30.Position := 0.0;
   AxisNuw.Axis[1..15].Pos30.Speed := 0;
   AxisNuw.Axis[1..15].Pos30.Reached := FALSE;
   AxisDisplay.Axis[1..15].Pos1.Position := 0.0;
   AxisDisplay.Axis[1..15].Pos1.Speed := 0;
   AxisDisplay.Axis[1..15].Pos1.Reached := FALSE;
   AxisDisplay.Axis[1..15].Pos2.Position := 0.0;
   AxisDisplay.Axis[1..15].Pos2.Speed := 0;
   AxisDisplay.Axis[1..15].Pos2.Reached := FALSE;
   AxisDisplay.Axis[1..15].Pos3.Position := 0.0;
   AxisDisplay.Axis[1..15].Pos3.Speed := 0;
   AxisDisplay.Axis[1..15].Pos3.Reached := FALSE;
   AxisDisplay.Axis[1..15].Pos4.Position := 0.0;
   AxisDisplay.Axis[1..15].Pos4.Speed := 0;
   AxisDisplay.Axis[1..15].Pos4.Reached := FALSE;
   AxisDisplay.Axis[1..15].Pos5.Position := 0.0;
   AxisDisplay.Axis[1..15].Pos5.Speed := 0;
   AxisDisplay.Axis[1..15].Pos5.Reached := FALSE;
   AxisDisplay.Axis[1..15].Pos6.Position := 0.0;
   AxisDisplay.Axis[1..15].Pos6.Speed := 0;
   AxisDisplay.Axis[1..15].Pos6.Reached := FALSE;
   AxisDisplay.Axis[1..15].Pos7.Position := 0.0;
   AxisDisplay.Axis[1..15].Pos7.Speed := 0;
   AxisDisplay.Axis[1..15].Pos7.Reached := FALSE;
   AxisDisplay.Axis[1..15].Pos8.Position := 0.0;
   AxisDisplay.Axis[1..15].Pos8.Speed := 0;
   AxisDisplay.Axis[1..15].Pos8.Reached := FALSE;
   AxisDisplay.Axis[1..15].Pos9.Position := 0.0;
   AxisDisplay.Axis[1..15].Pos9.Speed := 0;
   AxisDisplay.Axis[1..15].Pos9.Reached := FALSE;
   AxisDisplay.Axis[1..15].Pos10.Position := 0.0;
   AxisDisplay.Axis[1..15].Pos10.Speed := 0;
   AxisDisplay.Axis[1..15].Pos10.Reached := FALSE;
   AxisDisplay.Axis[1..15].Pos11.Position := 0.0;
   AxisDisplay.Axis[1..15].Pos11.Speed := 0;
   AxisDisplay.Axis[1..15].Pos11.Reached := FALSE;
   AxisDisplay.Axis[1..15].Pos12.Position := 0.0;
   AxisDisplay.Axis[1..15].Pos12.Speed := 0;
   AxisDisplay.Axis[1..15].Pos12.Reached := FALSE;
   AxisDisplay.Axis[1..15].Pos13.Position := 0.0;
   AxisDisplay.Axis[1..15].Pos13.Speed := 0;
   AxisDisplay.Axis[1..15].Pos13.Reached := FALSE;
   AxisDisplay.Axis[1..15].Pos14.Position := 0.0;
   AxisDisplay.Axis[1..15].Pos14.Speed := 0;
   AxisDisplay.Axis[1..15].Pos14.Reached := FALSE;
   AxisDisplay.Axis[1..15].Pos15.Position := 0.0;
   AxisDisplay.Axis[1..15].Pos15.Speed := 0;
   AxisDisplay.Axis[1..15].Pos15.Reached := FALSE;
   AxisDisplay.Axis[1..15].Pos16.Position := 0.0;
   AxisDisplay.Axis[1..15].Pos16.Speed := 0;
   AxisDisplay.Axis[1..15].Pos16.Reached := FALSE;
   AxisDisplay.Axis[1..15].Pos17.Position := 0.0;
   AxisDisplay.Axis[1..15].Pos17.Speed := 0;
   AxisDisplay.Axis[1..15].Pos17.Reached := FALSE;
   AxisDisplay.Axis[1..15].Pos18.Position := 0.0;
   AxisDisplay.Axis[1..15].Pos18.Speed := 0;
   AxisDisplay.Axis[1..15].Pos18.Reached := FALSE;
   AxisDisplay.Axis[1..15].Pos19.Position := 0.0;
   AxisDisplay.Axis[1..15].Pos19.Speed := 0;
   AxisDisplay.Axis[1..15].Pos19.Reached := FALSE;
   AxisDisplay.Axis[1..15].Pos20.Position := 0.0;
   AxisDisplay.Axis[1..15].Pos20.Speed := 0;
   AxisDisplay.Axis[1..15].Pos20.Reached := FALSE;
   AxisDisplay.Axis[1..15].Pos21.Position := 0.0;
   AxisDisplay.Axis[1..15].Pos21.Speed := 0;
   AxisDisplay.Axis[1..15].Pos21.Reached := FALSE;
   AxisDisplay.Axis[1..15].Pos22.Position := 0.0;
   AxisDisplay.Axis[1..15].Pos22.Speed := 0;
   AxisDisplay.Axis[1..15].Pos22.Reached := FALSE;
   AxisDisplay.Axis[1..15].Pos23.Position := 0.0;
   AxisDisplay.Axis[1..15].Pos23.Speed := 0;
   AxisDisplay.Axis[1..15].Pos23.Reached := FALSE;
   AxisDisplay.Axis[1..15].Pos24.Position := 0.0;
   AxisDisplay.Axis[1..15].Pos24.Speed := 0;
   AxisDisplay.Axis[1..15].Pos24.Reached := FALSE;
   AxisDisplay.Axis[1..15].Pos25.Position := 0.0;
   AxisDisplay.Axis[1..15].Pos25.Speed := 0;
   AxisDisplay.Axis[1..15].Pos25.Reached := FALSE;
   AxisDisplay.Axis[1..15].Pos26.Position := 0.0;
   AxisDisplay.Axis[1..15].Pos26.Speed := 0;
   AxisDisplay.Axis[1..15].Pos26.Reached := FALSE;
   AxisDisplay.Axis[1..15].Pos27.Position := 0.0;
   AxisDisplay.Axis[1..15].Pos27.Speed := 0;
   AxisDisplay.Axis[1..15].Pos27.Reached := FALSE;
   AxisDisplay.Axis[1..15].Pos28.Position := 0.0;
   AxisDisplay.Axis[1..15].Pos28.Speed := 0;
   AxisDisplay.Axis[1..15].Pos28.Reached := FALSE;
   AxisDisplay.Axis[1..15].Pos29.Position := 0.0;
   AxisDisplay.Axis[1..15].Pos29.Speed := 0;
   AxisDisplay.Axis[1..15].Pos29.Reached := FALSE;
   AxisDisplay.Axis[1..15].Pos30.Position := 0.0;
   AxisDisplay.Axis[1..15].Pos30.Speed := 0;
   AxisDisplay.Axis[1..15].Pos30.Reached := FALSE;
   AxisSave.Axis[1..15].Pos1.Position := 0.0;
   AxisSave.Axis[1..15].Pos1.Speed := 0;
   AxisSave.Axis[1..15].Pos1.Reached := FALSE;
   AxisSave.Axis[1..15].Pos2.Position := 0.0;
   AxisSave.Axis[1..15].Pos2.Speed := 0;
   AxisSave.Axis[1..15].Pos2.Reached := FALSE;
   AxisSave.Axis[1..15].Pos3.Position := 0.0;
   AxisSave.Axis[1..15].Pos3.Speed := 0;
   AxisSave.Axis[1..15].Pos3.Reached := FALSE;
   AxisSave.Axis[1..15].Pos4.Position := 0.0;
   AxisSave.Axis[1..15].Pos4.Speed := 0;
   AxisSave.Axis[1..15].Pos4.Reached := FALSE;
   AxisSave.Axis[1..15].Pos5.Position := 0.0;
   AxisSave.Axis[1..15].Pos5.Speed := 0;
   AxisSave.Axis[1..15].Pos5.Reached := FALSE;
   AxisSave.Axis[1..15].Pos6.Position := 0.0;
   AxisSave.Axis[1..15].Pos6.Speed := 0;
   AxisSave.Axis[1..15].Pos6.Reached := FALSE;
   AxisSave.Axis[1..15].Pos7.Position := 0.0;
   AxisSave.Axis[1..15].Pos7.Speed := 0;
   AxisSave.Axis[1..15].Pos7.Reached := FALSE;
   AxisSave.Axis[1..15].Pos8.Position := 0.0;
   AxisSave.Axis[1..15].Pos8.Speed := 0;
   AxisSave.Axis[1..15].Pos8.Reached := FALSE;
   AxisSave.Axis[1..15].Pos9.Position := 0.0;
   AxisSave.Axis[1..15].Pos9.Speed := 0;
   AxisSave.Axis[1..15].Pos9.Reached := FALSE;
   AxisSave.Axis[1..15].Pos10.Position := 0.0;
   AxisSave.Axis[1..15].Pos10.Speed := 0;
   AxisSave.Axis[1..15].Pos10.Reached := FALSE;
   AxisSave.Axis[1..15].Pos11.Position := 0.0;
   AxisSave.Axis[1..15].Pos11.Speed := 0;
   AxisSave.Axis[1..15].Pos11.Reached := FALSE;
   AxisSave.Axis[1..15].Pos12.Position := 0.0;
   AxisSave.Axis[1..15].Pos12.Speed := 0;
   AxisSave.Axis[1..15].Pos12.Reached := FALSE;
   AxisSave.Axis[1..15].Pos13.Position := 0.0;
   AxisSave.Axis[1..15].Pos13.Speed := 0;
   AxisSave.Axis[1..15].Pos13.Reached := FALSE;
   AxisSave.Axis[1..15].Pos14.Position := 0.0;
   AxisSave.Axis[1..15].Pos14.Speed := 0;
   AxisSave.Axis[1..15].Pos14.Reached := FALSE;
   AxisSave.Axis[1..15].Pos15.Position := 0.0;
   AxisSave.Axis[1..15].Pos15.Speed := 0;
   AxisSave.Axis[1..15].Pos15.Reached := FALSE;
   AxisSave.Axis[1..15].Pos16.Position := 0.0;
   AxisSave.Axis[1..15].Pos16.Speed := 0;
   AxisSave.Axis[1..15].Pos16.Reached := FALSE;
   AxisSave.Axis[1..15].Pos17.Position := 0.0;
   AxisSave.Axis[1..15].Pos17.Speed := 0;
   AxisSave.Axis[1..15].Pos17.Reached := FALSE;
   AxisSave.Axis[1..15].Pos18.Position := 0.0;
   AxisSave.Axis[1..15].Pos18.Speed := 0;
   AxisSave.Axis[1..15].Pos18.Reached := FALSE;
   AxisSave.Axis[1..15].Pos19.Position := 0.0;
   AxisSave.Axis[1..15].Pos19.Speed := 0;
   AxisSave.Axis[1..15].Pos19.Reached := FALSE;
   AxisSave.Axis[1..15].Pos20.Position := 0.0;
   AxisSave.Axis[1..15].Pos20.Speed := 0;
   AxisSave.Axis[1..15].Pos20.Reached := FALSE;
   AxisSave.Axis[1..15].Pos21.Position := 0.0;
   AxisSave.Axis[1..15].Pos21.Speed := 0;
   AxisSave.Axis[1..15].Pos21.Reached := FALSE;
   AxisSave.Axis[1..15].Pos22.Position := 0.0;
   AxisSave.Axis[1..15].Pos22.Speed := 0;
   AxisSave.Axis[1..15].Pos22.Reached := FALSE;
   AxisSave.Axis[1..15].Pos23.Position := 0.0;
   AxisSave.Axis[1..15].Pos23.Speed := 0;
   AxisSave.Axis[1..15].Pos23.Reached := FALSE;
   AxisSave.Axis[1..15].Pos24.Position := 0.0;
   AxisSave.Axis[1..15].Pos24.Speed := 0;
   AxisSave.Axis[1..15].Pos24.Reached := FALSE;
   AxisSave.Axis[1..15].Pos25.Position := 0.0;
   AxisSave.Axis[1..15].Pos25.Speed := 0;
   AxisSave.Axis[1..15].Pos25.Reached := FALSE;
   AxisSave.Axis[1..15].Pos26.Position := 0.0;
   AxisSave.Axis[1..15].Pos26.Speed := 0;
   AxisSave.Axis[1..15].Pos26.Reached := FALSE;
   AxisSave.Axis[1..15].Pos27.Position := 0.0;
   AxisSave.Axis[1..15].Pos27.Speed := 0;
   AxisSave.Axis[1..15].Pos27.Reached := FALSE;
   AxisSave.Axis[1..15].Pos28.Position := 0.0;
   AxisSave.Axis[1..15].Pos28.Speed := 0;
   AxisSave.Axis[1..15].Pos28.Reached := FALSE;
   AxisSave.Axis[1..15].Pos29.Position := 0.0;
   AxisSave.Axis[1..15].Pos29.Speed := 0;
   AxisSave.Axis[1..15].Pos29.Reached := FALSE;
   AxisSave.Axis[1..15].Pos30.Position := 0.0;
   AxisSave.Axis[1..15].Pos30.Speed := 0;
   AxisSave.Axis[1..15].Pos30.Reached := FALSE;
   AxisStore[1].Axis[1..15].Pos1.Position := 0.0;
   AxisStore[2].Axis[1..15].Pos1.Position := 0.0;
   AxisStore[3].Axis[1..15].Pos1.Position := 0.0;
   AxisStore[4].Axis[1..15].Pos1.Position := 0.0;
   AxisStore[5].Axis[1..15].Pos1.Position := 0.0;
   AxisStore[6].Axis[1..15].Pos1.Position := 0.0;
   AxisStore[7].Axis[1..15].Pos1.Position := 0.0;
   AxisStore[8].Axis[1..15].Pos1.Position := 0.0;
   AxisStore[9].Axis[1..15].Pos1.Position := 0.0;
   AxisStore[10].Axis[1..15].Pos1.Position := 0.0;
   AxisStore[11].Axis[1..15].Pos1.Position := 0.0;
   AxisStore[12].Axis[1..15].Pos1.Position := 0.0;
   AxisStore[13].Axis[1..15].Pos1.Position := 0.0;
   AxisStore[14].Axis[1..15].Pos1.Position := 0.0;
   AxisStore[15].Axis[1..15].Pos1.Position := 0.0;
   AxisStore[1].Axis[1..15].Pos1.Speed := 0;
   AxisStore[2].Axis[1..15].Pos1.Speed := 0;
   AxisStore[3].Axis[1..15].Pos1.Speed := 0;
   AxisStore[4].Axis[1..15].Pos1.Speed := 0;
   AxisStore[5].Axis[1..15].Pos1.Speed := 0;
   AxisStore[6].Axis[1..15].Pos1.Speed := 0;
   AxisStore[7].Axis[1..15].Pos1.Speed := 0;
   AxisStore[8].Axis[1..15].Pos1.Speed := 0;
   AxisStore[9].Axis[1..15].Pos1.Speed := 0;
   AxisStore[10].Axis[1..15].Pos1.Speed := 0;
   AxisStore[11].Axis[1..15].Pos1.Speed := 0;
   AxisStore[12].Axis[1..15].Pos1.Speed := 0;
   AxisStore[13].Axis[1..15].Pos1.Speed := 0;
   AxisStore[14].Axis[1..15].Pos1.Speed := 0;
   AxisStore[15].Axis[1..15].Pos1.Speed := 0;
   AxisStore[1].Axis[1..15].Pos1.Reached := FALSE;
   AxisStore[2].Axis[1..15].Pos1.Reached := FALSE;
   AxisStore[3].Axis[1..15].Pos1.Reached := FALSE;
   AxisStore[4].Axis[1..15].Pos1.Reached := FALSE;
   AxisStore[5].Axis[1..15].Pos1.Reached := FALSE;
   AxisStore[6].Axis[1..15].Pos1.Reached := FALSE;
   AxisStore[7].Axis[1..15].Pos1.Reached := FALSE;
   AxisStore[8].Axis[1..15].Pos1.Reached := FALSE;
   AxisStore[9].Axis[1..15].Pos1.Reached := FALSE;
   AxisStore[10].Axis[1..15].Pos1.Reached := FALSE;
   AxisStore[11].Axis[1..15].Pos1.Reached := FALSE;
   AxisStore[12].Axis[1..15].Pos1.Reached := FALSE;
   AxisStore[13].Axis[1..15].Pos1.Reached := FALSE;
   AxisStore[14].Axis[1..15].Pos1.Reached := FALSE;
   AxisStore[15].Axis[1..15].Pos1.Reached := FALSE;
   AxisStore[1].Axis[1..15].Pos2.Position := 0.0;
   AxisStore[2].Axis[1..15].Pos2.Position := 0.0;
   AxisStore[3].Axis[1..15].Pos2.Position := 0.0;
   AxisStore[4].Axis[1..15].Pos2.Position := 0.0;
   AxisStore[5].Axis[1..15].Pos2.Position := 0.0;
   AxisStore[6].Axis[1..15].Pos2.Position := 0.0;
   AxisStore[7].Axis[1..15].Pos2.Position := 0.0;
   AxisStore[8].Axis[1..15].Pos2.Position := 0.0;
   AxisStore[9].Axis[1..15].Pos2.Position := 0.0;
   AxisStore[10].Axis[1..15].Pos2.Position := 0.0;
   AxisStore[11].Axis[1..15].Pos2.Position := 0.0;
   AxisStore[12].Axis[1..15].Pos2.Position := 0.0;
   AxisStore[13].Axis[1..15].Pos2.Position := 0.0;
   AxisStore[14].Axis[1..15].Pos2.Position := 0.0;
   AxisStore[15].Axis[1..15].Pos2.Position := 0.0;
   AxisStore[1].Axis[1..15].Pos2.Speed := 0;
   AxisStore[2].Axis[1..15].Pos2.Speed := 0;
   AxisStore[3].Axis[1..15].Pos2.Speed := 0;
   AxisStore[4].Axis[1..15].Pos2.Speed := 0;
   AxisStore[5].Axis[1..15].Pos2.Speed := 0;
   AxisStore[6].Axis[1..15].Pos2.Speed := 0;
   AxisStore[7].Axis[1..15].Pos2.Speed := 0;
   AxisStore[8].Axis[1..15].Pos2.Speed := 0;
   AxisStore[9].Axis[1..15].Pos2.Speed := 0;
   AxisStore[10].Axis[1..15].Pos2.Speed := 0;
   AxisStore[11].Axis[1..15].Pos2.Speed := 0;
   AxisStore[12].Axis[1..15].Pos2.Speed := 0;
   AxisStore[13].Axis[1..15].Pos2.Speed := 0;
   AxisStore[14].Axis[1..15].Pos2.Speed := 0;
   AxisStore[15].Axis[1..15].Pos2.Speed := 0;
   AxisStore[1].Axis[1..15].Pos2.Reached := FALSE;
   AxisStore[2].Axis[1..15].Pos2.Reached := FALSE;
   AxisStore[3].Axis[1..15].Pos2.Reached := FALSE;
   AxisStore[4].Axis[1..15].Pos2.Reached := FALSE;
   AxisStore[5].Axis[1..15].Pos2.Reached := FALSE;
   AxisStore[6].Axis[1..15].Pos2.Reached := FALSE;
   AxisStore[7].Axis[1..15].Pos2.Reached := FALSE;
   AxisStore[8].Axis[1..15].Pos2.Reached := FALSE;
   AxisStore[9].Axis[1..15].Pos2.Reached := FALSE;
   AxisStore[10].Axis[1..15].Pos2.Reached := FALSE;
   AxisStore[11].Axis[1..15].Pos2.Reached := FALSE;
   AxisStore[12].Axis[1..15].Pos2.Reached := FALSE;
   AxisStore[13].Axis[1..15].Pos2.Reached := FALSE;
   AxisStore[14].Axis[1..15].Pos2.Reached := FALSE;
   AxisStore[15].Axis[1..15].Pos2.Reached := FALSE;
   AxisStore[1].Axis[1..15].Pos3.Position := 0.0;
   AxisStore[2].Axis[1..15].Pos3.Position := 0.0;
   AxisStore[3].Axis[1..15].Pos3.Position := 0.0;
   AxisStore[4].Axis[1..15].Pos3.Position := 0.0;
   AxisStore[5].Axis[1..15].Pos3.Position := 0.0;
   AxisStore[6].Axis[1..15].Pos3.Position := 0.0;
   AxisStore[7].Axis[1..15].Pos3.Position := 0.0;
   AxisStore[8].Axis[1..15].Pos3.Position := 0.0;
   AxisStore[9].Axis[1..15].Pos3.Position := 0.0;
   AxisStore[10].Axis[1..15].Pos3.Position := 0.0;
   AxisStore[11].Axis[1..15].Pos3.Position := 0.0;
   AxisStore[12].Axis[1..15].Pos3.Position := 0.0;
   AxisStore[13].Axis[1..15].Pos3.Position := 0.0;
   AxisStore[14].Axis[1..15].Pos3.Position := 0.0;
   AxisStore[15].Axis[1..15].Pos3.Position := 0.0;
   AxisStore[1].Axis[1..15].Pos3.Speed := 0;
   AxisStore[2].Axis[1..15].Pos3.Speed := 0;
   AxisStore[3].Axis[1..15].Pos3.Speed := 0;
   AxisStore[4].Axis[1..15].Pos3.Speed := 0;
   AxisStore[5].Axis[1..15].Pos3.Speed := 0;
   AxisStore[6].Axis[1..15].Pos3.Speed := 0;
   AxisStore[7].Axis[1..15].Pos3.Speed := 0;
   AxisStore[8].Axis[1..15].Pos3.Speed := 0;
   AxisStore[9].Axis[1..15].Pos3.Speed := 0;
   AxisStore[10].Axis[1..15].Pos3.Speed := 0;
   AxisStore[11].Axis[1..15].Pos3.Speed := 0;
   AxisStore[12].Axis[1..15].Pos3.Speed := 0;
   AxisStore[13].Axis[1..15].Pos3.Speed := 0;
   AxisStore[14].Axis[1..15].Pos3.Speed := 0;
   AxisStore[15].Axis[1..15].Pos3.Speed := 0;
   AxisStore[1].Axis[1..15].Pos3.Reached := FALSE;
   AxisStore[2].Axis[1..15].Pos3.Reached := FALSE;
   AxisStore[3].Axis[1..15].Pos3.Reached := FALSE;
   AxisStore[4].Axis[1..15].Pos3.Reached := FALSE;
   AxisStore[5].Axis[1..15].Pos3.Reached := FALSE;
   AxisStore[6].Axis[1..15].Pos3.Reached := FALSE;
   AxisStore[7].Axis[1..15].Pos3.Reached := FALSE;
   AxisStore[8].Axis[1..15].Pos3.Reached := FALSE;
   AxisStore[9].Axis[1..15].Pos3.Reached := FALSE;
   AxisStore[10].Axis[1..15].Pos3.Reached := FALSE;
   AxisStore[11].Axis[1..15].Pos3.Reached := FALSE;
   AxisStore[12].Axis[1..15].Pos3.Reached := FALSE;
   AxisStore[13].Axis[1..15].Pos3.Reached := FALSE;
   AxisStore[14].Axis[1..15].Pos3.Reached := FALSE;
   AxisStore[15].Axis[1..15].Pos3.Reached := FALSE;
   AxisStore[1].Axis[1..15].Pos4.Position := 0.0;
   AxisStore[2].Axis[1..15].Pos4.Position := 0.0;
   AxisStore[3].Axis[1..15].Pos4.Position := 0.0;
   AxisStore[4].Axis[1..15].Pos4.Position := 0.0;
   AxisStore[5].Axis[1..15].Pos4.Position := 0.0;
   AxisStore[6].Axis[1..15].Pos4.Position := 0.0;
   AxisStore[7].Axis[1..15].Pos4.Position := 0.0;
   AxisStore[8].Axis[1..15].Pos4.Position := 0.0;
   AxisStore[9].Axis[1..15].Pos4.Position := 0.0;
   AxisStore[10].Axis[1..15].Pos4.Position := 0.0;
   AxisStore[11].Axis[1..15].Pos4.Position := 0.0;
   AxisStore[12].Axis[1..15].Pos4.Position := 0.0;
   AxisStore[13].Axis[1..15].Pos4.Position := 0.0;
   AxisStore[14].Axis[1..15].Pos4.Position := 0.0;
   AxisStore[15].Axis[1..15].Pos4.Position := 0.0;
   AxisStore[1].Axis[1..15].Pos4.Speed := 0;
   AxisStore[2].Axis[1..15].Pos4.Speed := 0;
   AxisStore[3].Axis[1..15].Pos4.Speed := 0;
   AxisStore[4].Axis[1..15].Pos4.Speed := 0;
   AxisStore[5].Axis[1..15].Pos4.Speed := 0;
   AxisStore[6].Axis[1..15].Pos4.Speed := 0;
   AxisStore[7].Axis[1..15].Pos4.Speed := 0;
   AxisStore[8].Axis[1..15].Pos4.Speed := 0;
   AxisStore[9].Axis[1..15].Pos4.Speed := 0;
   AxisStore[10].Axis[1..15].Pos4.Speed := 0;
   AxisStore[11].Axis[1..15].Pos4.Speed := 0;
   AxisStore[12].Axis[1..15].Pos4.Speed := 0;
   AxisStore[13].Axis[1..15].Pos4.Speed := 0;
   AxisStore[14].Axis[1..15].Pos4.Speed := 0;
   AxisStore[15].Axis[1..15].Pos4.Speed := 0;
   AxisStore[1].Axis[1..15].Pos4.Reached := FALSE;
   AxisStore[2].Axis[1..15].Pos4.Reached := FALSE;
   AxisStore[3].Axis[1..15].Pos4.Reached := FALSE;
   AxisStore[4].Axis[1..15].Pos4.Reached := FALSE;
   AxisStore[5].Axis[1..15].Pos4.Reached := FALSE;
   AxisStore[6].Axis[1..15].Pos4.Reached := FALSE;
   AxisStore[7].Axis[1..15].Pos4.Reached := FALSE;
   AxisStore[8].Axis[1..15].Pos4.Reached := FALSE;
   AxisStore[9].Axis[1..15].Pos4.Reached := FALSE;
   AxisStore[10].Axis[1..15].Pos4.Reached := FALSE;
   AxisStore[11].Axis[1..15].Pos4.Reached := FALSE;
   AxisStore[12].Axis[1..15].Pos4.Reached := FALSE;
   AxisStore[13].Axis[1..15].Pos4.Reached := FALSE;
   AxisStore[14].Axis[1..15].Pos4.Reached := FALSE;
   AxisStore[15].Axis[1..15].Pos4.Reached := FALSE;
   AxisStore[1].Axis[1..15].Pos5.Position := 0.0;
   AxisStore[2].Axis[1..15].Pos5.Position := 0.0;
   AxisStore[3].Axis[1..15].Pos5.Position := 0.0;
   AxisStore[4].Axis[1..15].Pos5.Position := 0.0;
   AxisStore[5].Axis[1..15].Pos5.Position := 0.0;
   AxisStore[6].Axis[1..15].Pos5.Position := 0.0;
   AxisStore[7].Axis[1..15].Pos5.Position := 0.0;
   AxisStore[8].Axis[1..15].Pos5.Position := 0.0;
   AxisStore[9].Axis[1..15].Pos5.Position := 0.0;
   AxisStore[10].Axis[1..15].Pos5.Position := 0.0;
   AxisStore[11].Axis[1..15].Pos5.Position := 0.0;
   AxisStore[12].Axis[1..15].Pos5.Position := 0.0;
   AxisStore[13].Axis[1..15].Pos5.Position := 0.0;
   AxisStore[14].Axis[1..15].Pos5.Position := 0.0;
   AxisStore[15].Axis[1..15].Pos5.Position := 0.0;
   AxisStore[1].Axis[1..15].Pos5.Speed := 0;
   AxisStore[2].Axis[1..15].Pos5.Speed := 0;
   AxisStore[3].Axis[1..15].Pos5.Speed := 0;
   AxisStore[4].Axis[1..15].Pos5.Speed := 0;
   AxisStore[5].Axis[1..15].Pos5.Speed := 0;
   AxisStore[6].Axis[1..15].Pos5.Speed := 0;
   AxisStore[7].Axis[1..15].Pos5.Speed := 0;
   AxisStore[8].Axis[1..15].Pos5.Speed := 0;
   AxisStore[9].Axis[1..15].Pos5.Speed := 0;
   AxisStore[10].Axis[1..15].Pos5.Speed := 0;
   AxisStore[11].Axis[1..15].Pos5.Speed := 0;
   AxisStore[12].Axis[1..15].Pos5.Speed := 0;
   AxisStore[13].Axis[1..15].Pos5.Speed := 0;
   AxisStore[14].Axis[1..15].Pos5.Speed := 0;
   AxisStore[15].Axis[1..15].Pos5.Speed := 0;
   AxisStore[1].Axis[1..15].Pos5.Reached := FALSE;
   AxisStore[2].Axis[1..15].Pos5.Reached := FALSE;
   AxisStore[3].Axis[1..15].Pos5.Reached := FALSE;
   AxisStore[4].Axis[1..15].Pos5.Reached := FALSE;
   AxisStore[5].Axis[1..15].Pos5.Reached := FALSE;
   AxisStore[6].Axis[1..15].Pos5.Reached := FALSE;
   AxisStore[7].Axis[1..15].Pos5.Reached := FALSE;
   AxisStore[8].Axis[1..15].Pos5.Reached := FALSE;
   AxisStore[9].Axis[1..15].Pos5.Reached := FALSE;
   AxisStore[10].Axis[1..15].Pos5.Reached := FALSE;
   AxisStore[11].Axis[1..15].Pos5.Reached := FALSE;
   AxisStore[12].Axis[1..15].Pos5.Reached := FALSE;
   AxisStore[13].Axis[1..15].Pos5.Reached := FALSE;
   AxisStore[14].Axis[1..15].Pos5.Reached := FALSE;
   AxisStore[15].Axis[1..15].Pos5.Reached := FALSE;
   AxisStore[1].Axis[1..15].Pos6.Position := 0.0;
   AxisStore[2].Axis[1..15].Pos6.Position := 0.0;
   AxisStore[3].Axis[1..15].Pos6.Position := 0.0;
   AxisStore[4].Axis[1..15].Pos6.Position := 0.0;
   AxisStore[5].Axis[1..15].Pos6.Position := 0.0;
   AxisStore[6].Axis[1..15].Pos6.Position := 0.0;
   AxisStore[7].Axis[1..15].Pos6.Position := 0.0;
   AxisStore[8].Axis[1..15].Pos6.Position := 0.0;
   AxisStore[9].Axis[1..15].Pos6.Position := 0.0;
   AxisStore[10].Axis[1..15].Pos6.Position := 0.0;
   AxisStore[11].Axis[1..15].Pos6.Position := 0.0;
   AxisStore[12].Axis[1..15].Pos6.Position := 0.0;
   AxisStore[13].Axis[1..15].Pos6.Position := 0.0;
   AxisStore[14].Axis[1..15].Pos6.Position := 0.0;
   AxisStore[15].Axis[1..15].Pos6.Position := 0.0;
   AxisStore[1].Axis[1..15].Pos6.Speed := 0;
   AxisStore[2].Axis[1..15].Pos6.Speed := 0;
   AxisStore[3].Axis[1..15].Pos6.Speed := 0;
   AxisStore[4].Axis[1..15].Pos6.Speed := 0;
   AxisStore[5].Axis[1..15].Pos6.Speed := 0;
   AxisStore[6].Axis[1..15].Pos6.Speed := 0;
   AxisStore[7].Axis[1..15].Pos6.Speed := 0;
   AxisStore[8].Axis[1..15].Pos6.Speed := 0;
   AxisStore[9].Axis[1..15].Pos6.Speed := 0;
   AxisStore[10].Axis[1..15].Pos6.Speed := 0;
   AxisStore[11].Axis[1..15].Pos6.Speed := 0;
   AxisStore[12].Axis[1..15].Pos6.Speed := 0;
   AxisStore[13].Axis[1..15].Pos6.Speed := 0;
   AxisStore[14].Axis[1..15].Pos6.Speed := 0;
   AxisStore[15].Axis[1..15].Pos6.Speed := 0;
   AxisStore[1].Axis[1..15].Pos6.Reached := FALSE;
   AxisStore[2].Axis[1..15].Pos6.Reached := FALSE;
   AxisStore[3].Axis[1..15].Pos6.Reached := FALSE;
   AxisStore[4].Axis[1..15].Pos6.Reached := FALSE;
   AxisStore[5].Axis[1..15].Pos6.Reached := FALSE;
   AxisStore[6].Axis[1..15].Pos6.Reached := FALSE;
   AxisStore[7].Axis[1..15].Pos6.Reached := FALSE;
   AxisStore[8].Axis[1..15].Pos6.Reached := FALSE;
   AxisStore[9].Axis[1..15].Pos6.Reached := FALSE;
   AxisStore[10].Axis[1..15].Pos6.Reached := FALSE;
   AxisStore[11].Axis[1..15].Pos6.Reached := FALSE;
   AxisStore[12].Axis[1..15].Pos6.Reached := FALSE;
   AxisStore[13].Axis[1..15].Pos6.Reached := FALSE;
   AxisStore[14].Axis[1..15].Pos6.Reached := FALSE;
   AxisStore[15].Axis[1..15].Pos6.Reached := FALSE;
   AxisStore[1].Axis[1..15].Pos7.Position := 0.0;
   AxisStore[2].Axis[1..15].Pos7.Position := 0.0;
   AxisStore[3].Axis[1..15].Pos7.Position := 0.0;
   AxisStore[4].Axis[1..15].Pos7.Position := 0.0;
   AxisStore[5].Axis[1..15].Pos7.Position := 0.0;
   AxisStore[6].Axis[1..15].Pos7.Position := 0.0;
   AxisStore[7].Axis[1..15].Pos7.Position := 0.0;
   AxisStore[8].Axis[1..15].Pos7.Position := 0.0;
   AxisStore[9].Axis[1..15].Pos7.Position := 0.0;
   AxisStore[10].Axis[1..15].Pos7.Position := 0.0;
   AxisStore[11].Axis[1..15].Pos7.Position := 0.0;
   AxisStore[12].Axis[1..15].Pos7.Position := 0.0;
   AxisStore[13].Axis[1..15].Pos7.Position := 0.0;
   AxisStore[14].Axis[1..15].Pos7.Position := 0.0;
   AxisStore[15].Axis[1..15].Pos7.Position := 0.0;
   AxisStore[1].Axis[1..15].Pos7.Speed := 0;
   AxisStore[2].Axis[1..15].Pos7.Speed := 0;
   AxisStore[3].Axis[1..15].Pos7.Speed := 0;
   AxisStore[4].Axis[1..15].Pos7.Speed := 0;
   AxisStore[5].Axis[1..15].Pos7.Speed := 0;
   AxisStore[6].Axis[1..15].Pos7.Speed := 0;
   AxisStore[7].Axis[1..15].Pos7.Speed := 0;
   AxisStore[8].Axis[1..15].Pos7.Speed := 0;
   AxisStore[9].Axis[1..15].Pos7.Speed := 0;
   AxisStore[10].Axis[1..15].Pos7.Speed := 0;
   AxisStore[11].Axis[1..15].Pos7.Speed := 0;
   AxisStore[12].Axis[1..15].Pos7.Speed := 0;
   AxisStore[13].Axis[1..15].Pos7.Speed := 0;
   AxisStore[14].Axis[1..15].Pos7.Speed := 0;
   AxisStore[15].Axis[1..15].Pos7.Speed := 0;
   AxisStore[1].Axis[1..15].Pos7.Reached := FALSE;
   AxisStore[2].Axis[1..15].Pos7.Reached := FALSE;
   AxisStore[3].Axis[1..15].Pos7.Reached := FALSE;
   AxisStore[4].Axis[1..15].Pos7.Reached := FALSE;
   AxisStore[5].Axis[1..15].Pos7.Reached := FALSE;
   AxisStore[6].Axis[1..15].Pos7.Reached := FALSE;
   AxisStore[7].Axis[1..15].Pos7.Reached := FALSE;
   AxisStore[8].Axis[1..15].Pos7.Reached := FALSE;
   AxisStore[9].Axis[1..15].Pos7.Reached := FALSE;
   AxisStore[10].Axis[1..15].Pos7.Reached := FALSE;
   AxisStore[11].Axis[1..15].Pos7.Reached := FALSE;
   AxisStore[12].Axis[1..15].Pos7.Reached := FALSE;
   AxisStore[13].Axis[1..15].Pos7.Reached := FALSE;
   AxisStore[14].Axis[1..15].Pos7.Reached := FALSE;
   AxisStore[15].Axis[1..15].Pos7.Reached := FALSE;
   AxisStore[1].Axis[1..15].Pos8.Position := 0.0;
   AxisStore[2].Axis[1..15].Pos8.Position := 0.0;
   AxisStore[3].Axis[1..15].Pos8.Position := 0.0;
   AxisStore[4].Axis[1..15].Pos8.Position := 0.0;
   AxisStore[5].Axis[1..15].Pos8.Position := 0.0;
   AxisStore[6].Axis[1..15].Pos8.Position := 0.0;
   AxisStore[7].Axis[1..15].Pos8.Position := 0.0;
   AxisStore[8].Axis[1..15].Pos8.Position := 0.0;
   AxisStore[9].Axis[1..15].Pos8.Position := 0.0;
   AxisStore[10].Axis[1..15].Pos8.Position := 0.0;
   AxisStore[11].Axis[1..15].Pos8.Position := 0.0;
   AxisStore[12].Axis[1..15].Pos8.Position := 0.0;
   AxisStore[13].Axis[1..15].Pos8.Position := 0.0;
   AxisStore[14].Axis[1..15].Pos8.Position := 0.0;
   AxisStore[15].Axis[1..15].Pos8.Position := 0.0;
   AxisStore[1].Axis[1..15].Pos8.Speed := 0;
   AxisStore[2].Axis[1..15].Pos8.Speed := 0;
   AxisStore[3].Axis[1..15].Pos8.Speed := 0;
   AxisStore[4].Axis[1..15].Pos8.Speed := 0;
   AxisStore[5].Axis[1..15].Pos8.Speed := 0;
   AxisStore[6].Axis[1..15].Pos8.Speed := 0;
   AxisStore[7].Axis[1..15].Pos8.Speed := 0;
   AxisStore[8].Axis[1..15].Pos8.Speed := 0;
   AxisStore[9].Axis[1..15].Pos8.Speed := 0;
   AxisStore[10].Axis[1..15].Pos8.Speed := 0;
   AxisStore[11].Axis[1..15].Pos8.Speed := 0;
   AxisStore[12].Axis[1..15].Pos8.Speed := 0;
   AxisStore[13].Axis[1..15].Pos8.Speed := 0;
   AxisStore[14].Axis[1..15].Pos8.Speed := 0;
   AxisStore[15].Axis[1..15].Pos8.Speed := 0;
   AxisStore[1].Axis[1..15].Pos8.Reached := FALSE;
   AxisStore[2].Axis[1..15].Pos8.Reached := FALSE;
   AxisStore[3].Axis[1..15].Pos8.Reached := FALSE;
   AxisStore[4].Axis[1..15].Pos8.Reached := FALSE;
   AxisStore[5].Axis[1..15].Pos8.Reached := FALSE;
   AxisStore[6].Axis[1..15].Pos8.Reached := FALSE;
   AxisStore[7].Axis[1..15].Pos8.Reached := FALSE;
   AxisStore[8].Axis[1..15].Pos8.Reached := FALSE;
   AxisStore[9].Axis[1..15].Pos8.Reached := FALSE;
   AxisStore[10].Axis[1..15].Pos8.Reached := FALSE;
   AxisStore[11].Axis[1..15].Pos8.Reached := FALSE;
   AxisStore[12].Axis[1..15].Pos8.Reached := FALSE;
   AxisStore[13].Axis[1..15].Pos8.Reached := FALSE;
   AxisStore[14].Axis[1..15].Pos8.Reached := FALSE;
   AxisStore[15].Axis[1..15].Pos8.Reached := FALSE;
   AxisStore[1].Axis[1..15].Pos9.Position := 0.0;
   AxisStore[2].Axis[1..15].Pos9.Position := 0.0;
   AxisStore[3].Axis[1..15].Pos9.Position := 0.0;
   AxisStore[4].Axis[1..15].Pos9.Position := 0.0;
   AxisStore[5].Axis[1..15].Pos9.Position := 0.0;
   AxisStore[6].Axis[1..15].Pos9.Position := 0.0;
   AxisStore[7].Axis[1..15].Pos9.Position := 0.0;
   AxisStore[8].Axis[1..15].Pos9.Position := 0.0;
   AxisStore[9].Axis[1..15].Pos9.Position := 0.0;
   AxisStore[10].Axis[1..15].Pos9.Position := 0.0;
   AxisStore[11].Axis[1..15].Pos9.Position := 0.0;
   AxisStore[12].Axis[1..15].Pos9.Position := 0.0;
   AxisStore[13].Axis[1..15].Pos9.Position := 0.0;
   AxisStore[14].Axis[1..15].Pos9.Position := 0.0;
   AxisStore[15].Axis[1..15].Pos9.Position := 0.0;
   AxisStore[1].Axis[1..15].Pos9.Speed := 0;
   AxisStore[2].Axis[1..15].Pos9.Speed := 0;
   AxisStore[3].Axis[1..15].Pos9.Speed := 0;
   AxisStore[4].Axis[1..15].Pos9.Speed := 0;
   AxisStore[5].Axis[1..15].Pos9.Speed := 0;
   AxisStore[6].Axis[1..15].Pos9.Speed := 0;
   AxisStore[7].Axis[1..15].Pos9.Speed := 0;
   AxisStore[8].Axis[1..15].Pos9.Speed := 0;
   AxisStore[9].Axis[1..15].Pos9.Speed := 0;
   AxisStore[10].Axis[1..15].Pos9.Speed := 0;
   AxisStore[11].Axis[1..15].Pos9.Speed := 0;
   AxisStore[12].Axis[1..15].Pos9.Speed := 0;
   AxisStore[13].Axis[1..15].Pos9.Speed := 0;
   AxisStore[14].Axis[1..15].Pos9.Speed := 0;
   AxisStore[15].Axis[1..15].Pos9.Speed := 0;
   AxisStore[1].Axis[1..15].Pos9.Reached := FALSE;
   AxisStore[2].Axis[1..15].Pos9.Reached := FALSE;
   AxisStore[3].Axis[1..15].Pos9.Reached := FALSE;
   AxisStore[4].Axis[1..15].Pos9.Reached := FALSE;
   AxisStore[5].Axis[1..15].Pos9.Reached := FALSE;
   AxisStore[6].Axis[1..15].Pos9.Reached := FALSE;
   AxisStore[7].Axis[1..15].Pos9.Reached := FALSE;
   AxisStore[8].Axis[1..15].Pos9.Reached := FALSE;
   AxisStore[9].Axis[1..15].Pos9.Reached := FALSE;
   AxisStore[10].Axis[1..15].Pos9.Reached := FALSE;
   AxisStore[11].Axis[1..15].Pos9.Reached := FALSE;
   AxisStore[12].Axis[1..15].Pos9.Reached := FALSE;
   AxisStore[13].Axis[1..15].Pos9.Reached := FALSE;
   AxisStore[14].Axis[1..15].Pos9.Reached := FALSE;
   AxisStore[15].Axis[1..15].Pos9.Reached := FALSE;
   AxisStore[1].Axis[1..15].Pos10.Position := 0.0;
   AxisStore[2].Axis[1..15].Pos10.Position := 0.0;
   AxisStore[3].Axis[1..15].Pos10.Position := 0.0;
   AxisStore[4].Axis[1..15].Pos10.Position := 0.0;
   AxisStore[5].Axis[1..15].Pos10.Position := 0.0;
   AxisStore[6].Axis[1..15].Pos10.Position := 0.0;
   AxisStore[7].Axis[1..15].Pos10.Position := 0.0;
   AxisStore[8].Axis[1..15].Pos10.Position := 0.0;
   AxisStore[9].Axis[1..15].Pos10.Position := 0.0;
   AxisStore[10].Axis[1..15].Pos10.Position := 0.0;
   AxisStore[11].Axis[1..15].Pos10.Position := 0.0;
   AxisStore[12].Axis[1..15].Pos10.Position := 0.0;
   AxisStore[13].Axis[1..15].Pos10.Position := 0.0;
   AxisStore[14].Axis[1..15].Pos10.Position := 0.0;
   AxisStore[15].Axis[1..15].Pos10.Position := 0.0;
   AxisStore[1].Axis[1..15].Pos10.Speed := 0;
   AxisStore[2].Axis[1..15].Pos10.Speed := 0;
   AxisStore[3].Axis[1..15].Pos10.Speed := 0;
   AxisStore[4].Axis[1..15].Pos10.Speed := 0;
   AxisStore[5].Axis[1..15].Pos10.Speed := 0;
   AxisStore[6].Axis[1..15].Pos10.Speed := 0;
   AxisStore[7].Axis[1..15].Pos10.Speed := 0;
   AxisStore[8].Axis[1..15].Pos10.Speed := 0;
   AxisStore[9].Axis[1..15].Pos10.Speed := 0;
   AxisStore[10].Axis[1..15].Pos10.Speed := 0;
   AxisStore[11].Axis[1..15].Pos10.Speed := 0;
   AxisStore[12].Axis[1..15].Pos10.Speed := 0;
   AxisStore[13].Axis[1..15].Pos10.Speed := 0;
   AxisStore[14].Axis[1..15].Pos10.Speed := 0;
   AxisStore[15].Axis[1..15].Pos10.Speed := 0;
   AxisStore[1].Axis[1..15].Pos10.Reached := FALSE;
   AxisStore[2].Axis[1..15].Pos10.Reached := FALSE;
   AxisStore[3].Axis[1..15].Pos10.Reached := FALSE;
   AxisStore[4].Axis[1..15].Pos10.Reached := FALSE;
   AxisStore[5].Axis[1..15].Pos10.Reached := FALSE;
   AxisStore[6].Axis[1..15].Pos10.Reached := FALSE;
   AxisStore[7].Axis[1..15].Pos10.Reached := FALSE;
   AxisStore[8].Axis[1..15].Pos10.Reached := FALSE;
   AxisStore[9].Axis[1..15].Pos10.Reached := FALSE;
   AxisStore[10].Axis[1..15].Pos10.Reached := FALSE;
   AxisStore[11].Axis[1..15].Pos10.Reached := FALSE;
   AxisStore[12].Axis[1..15].Pos10.Reached := FALSE;
   AxisStore[13].Axis[1..15].Pos10.Reached := FALSE;
   AxisStore[14].Axis[1..15].Pos10.Reached := FALSE;
   AxisStore[15].Axis[1..15].Pos10.Reached := FALSE;
   AxisStore[1].Axis[1..15].Pos11.Position := 0.0;
   AxisStore[2].Axis[1..15].Pos11.Position := 0.0;
   AxisStore[3].Axis[1..15].Pos11.Position := 0.0;
   AxisStore[4].Axis[1..15].Pos11.Position := 0.0;
   AxisStore[5].Axis[1..15].Pos11.Position := 0.0;
   AxisStore[6].Axis[1..15].Pos11.Position := 0.0;
   AxisStore[7].Axis[1..15].Pos11.Position := 0.0;
   AxisStore[8].Axis[1..15].Pos11.Position := 0.0;
   AxisStore[9].Axis[1..15].Pos11.Position := 0.0;
   AxisStore[10].Axis[1..15].Pos11.Position := 0.0;
   AxisStore[11].Axis[1..15].Pos11.Position := 0.0;
   AxisStore[12].Axis[1..15].Pos11.Position := 0.0;
   AxisStore[13].Axis[1..15].Pos11.Position := 0.0;
   AxisStore[14].Axis[1..15].Pos11.Position := 0.0;
   AxisStore[15].Axis[1..15].Pos11.Position := 0.0;
   AxisStore[1].Axis[1..15].Pos11.Speed := 0;
   AxisStore[2].Axis[1..15].Pos11.Speed := 0;
   AxisStore[3].Axis[1..15].Pos11.Speed := 0;
   AxisStore[4].Axis[1..15].Pos11.Speed := 0;
   AxisStore[5].Axis[1..15].Pos11.Speed := 0;
   AxisStore[6].Axis[1..15].Pos11.Speed := 0;
   AxisStore[7].Axis[1..15].Pos11.Speed := 0;
   AxisStore[8].Axis[1..15].Pos11.Speed := 0;
   AxisStore[9].Axis[1..15].Pos11.Speed := 0;
   AxisStore[10].Axis[1..15].Pos11.Speed := 0;
   AxisStore[11].Axis[1..15].Pos11.Speed := 0;
   AxisStore[12].Axis[1..15].Pos11.Speed := 0;
   AxisStore[13].Axis[1..15].Pos11.Speed := 0;
   AxisStore[14].Axis[1..15].Pos11.Speed := 0;
   AxisStore[15].Axis[1..15].Pos11.Speed := 0;
   AxisStore[1].Axis[1..15].Pos11.Reached := FALSE;
   AxisStore[2].Axis[1..15].Pos11.Reached := FALSE;
   AxisStore[3].Axis[1..15].Pos11.Reached := FALSE;
   AxisStore[4].Axis[1..15].Pos11.Reached := FALSE;
   AxisStore[5].Axis[1..15].Pos11.Reached := FALSE;
   AxisStore[6].Axis[1..15].Pos11.Reached := FALSE;
   AxisStore[7].Axis[1..15].Pos11.Reached := FALSE;
   AxisStore[8].Axis[1..15].Pos11.Reached := FALSE;
   AxisStore[9].Axis[1..15].Pos11.Reached := FALSE;
   AxisStore[10].Axis[1..15].Pos11.Reached := FALSE;
   AxisStore[11].Axis[1..15].Pos11.Reached := FALSE;
   AxisStore[12].Axis[1..15].Pos11.Reached := FALSE;
   AxisStore[13].Axis[1..15].Pos11.Reached := FALSE;
   AxisStore[14].Axis[1..15].Pos11.Reached := FALSE;
   AxisStore[15].Axis[1..15].Pos11.Reached := FALSE;
   AxisStore[1].Axis[1..15].Pos12.Position := 0.0;
   AxisStore[2].Axis[1..15].Pos12.Position := 0.0;
   AxisStore[3].Axis[1..15].Pos12.Position := 0.0;
   AxisStore[4].Axis[1..15].Pos12.Position := 0.0;
   AxisStore[5].Axis[1..15].Pos12.Position := 0.0;
   AxisStore[6].Axis[1..15].Pos12.Position := 0.0;
   AxisStore[7].Axis[1..15].Pos12.Position := 0.0;
   AxisStore[8].Axis[1..15].Pos12.Position := 0.0;
   AxisStore[9].Axis[1..15].Pos12.Position := 0.0;
   AxisStore[10].Axis[1..15].Pos12.Position := 0.0;
   AxisStore[11].Axis[1..15].Pos12.Position := 0.0;
   AxisStore[12].Axis[1..15].Pos12.Position := 0.0;
   AxisStore[13].Axis[1..15].Pos12.Position := 0.0;
   AxisStore[14].Axis[1..15].Pos12.Position := 0.0;
   AxisStore[15].Axis[1..15].Pos12.Position := 0.0;
   AxisStore[1].Axis[1..15].Pos12.Speed := 0;
   AxisStore[2].Axis[1..15].Pos12.Speed := 0;
   AxisStore[3].Axis[1..15].Pos12.Speed := 0;
   AxisStore[4].Axis[1..15].Pos12.Speed := 0;
   AxisStore[5].Axis[1..15].Pos12.Speed := 0;
   AxisStore[6].Axis[1..15].Pos12.Speed := 0;
   AxisStore[7].Axis[1..15].Pos12.Speed := 0;
   AxisStore[8].Axis[1..15].Pos12.Speed := 0;
   AxisStore[9].Axis[1..15].Pos12.Speed := 0;
   AxisStore[10].Axis[1..15].Pos12.Speed := 0;
   AxisStore[11].Axis[1..15].Pos12.Speed := 0;
   AxisStore[12].Axis[1..15].Pos12.Speed := 0;
   AxisStore[13].Axis[1..15].Pos12.Speed := 0;
   AxisStore[14].Axis[1..15].Pos12.Speed := 0;
   AxisStore[15].Axis[1..15].Pos12.Speed := 0;
   AxisStore[1].Axis[1..15].Pos12.Reached := FALSE;
   AxisStore[2].Axis[1..15].Pos12.Reached := FALSE;
   AxisStore[3].Axis[1..15].Pos12.Reached := FALSE;
   AxisStore[4].Axis[1..15].Pos12.Reached := FALSE;
   AxisStore[5].Axis[1..15].Pos12.Reached := FALSE;
   AxisStore[6].Axis[1..15].Pos12.Reached := FALSE;
   AxisStore[7].Axis[1..15].Pos12.Reached := FALSE;
   AxisStore[8].Axis[1..15].Pos12.Reached := FALSE;
   AxisStore[9].Axis[1..15].Pos12.Reached := FALSE;
   AxisStore[10].Axis[1..15].Pos12.Reached := FALSE;
   AxisStore[11].Axis[1..15].Pos12.Reached := FALSE;
   AxisStore[12].Axis[1..15].Pos12.Reached := FALSE;
   AxisStore[13].Axis[1..15].Pos12.Reached := FALSE;
   AxisStore[14].Axis[1..15].Pos12.Reached := FALSE;
   AxisStore[15].Axis[1..15].Pos12.Reached := FALSE;
   AxisStore[1].Axis[1..15].Pos13.Position := 0.0;
   AxisStore[2].Axis[1..15].Pos13.Position := 0.0;
   AxisStore[3].Axis[1..15].Pos13.Position := 0.0;
   AxisStore[4].Axis[1..15].Pos13.Position := 0.0;
   AxisStore[5].Axis[1..15].Pos13.Position := 0.0;
   AxisStore[6].Axis[1..15].Pos13.Position := 0.0;
   AxisStore[7].Axis[1..15].Pos13.Position := 0.0;
   AxisStore[8].Axis[1..15].Pos13.Position := 0.0;
   AxisStore[9].Axis[1..15].Pos13.Position := 0.0;
   AxisStore[10].Axis[1..15].Pos13.Position := 0.0;
   AxisStore[11].Axis[1..15].Pos13.Position := 0.0;
   AxisStore[12].Axis[1..15].Pos13.Position := 0.0;
   AxisStore[13].Axis[1..15].Pos13.Position := 0.0;
   AxisStore[14].Axis[1..15].Pos13.Position := 0.0;
   AxisStore[15].Axis[1..15].Pos13.Position := 0.0;
   AxisStore[1].Axis[1..15].Pos13.Speed := 0;
   AxisStore[2].Axis[1..15].Pos13.Speed := 0;
   AxisStore[3].Axis[1..15].Pos13.Speed := 0;
   AxisStore[4].Axis[1..15].Pos13.Speed := 0;
   AxisStore[5].Axis[1..15].Pos13.Speed := 0;
   AxisStore[6].Axis[1..15].Pos13.Speed := 0;
   AxisStore[7].Axis[1..15].Pos13.Speed := 0;
   AxisStore[8].Axis[1..15].Pos13.Speed := 0;
   AxisStore[9].Axis[1..15].Pos13.Speed := 0;
   AxisStore[10].Axis[1..15].Pos13.Speed := 0;
   AxisStore[11].Axis[1..15].Pos13.Speed := 0;
   AxisStore[12].Axis[1..15].Pos13.Speed := 0;
   AxisStore[13].Axis[1..15].Pos13.Speed := 0;
   AxisStore[14].Axis[1..15].Pos13.Speed := 0;
   AxisStore[15].Axis[1..15].Pos13.Speed := 0;
   AxisStore[1].Axis[1..15].Pos13.Reached := FALSE;
   AxisStore[2].Axis[1..15].Pos13.Reached := FALSE;
   AxisStore[3].Axis[1..15].Pos13.Reached := FALSE;
   AxisStore[4].Axis[1..15].Pos13.Reached := FALSE;
   AxisStore[5].Axis[1..15].Pos13.Reached := FALSE;
   AxisStore[6].Axis[1..15].Pos13.Reached := FALSE;
   AxisStore[7].Axis[1..15].Pos13.Reached := FALSE;
   AxisStore[8].Axis[1..15].Pos13.Reached := FALSE;
   AxisStore[9].Axis[1..15].Pos13.Reached := FALSE;
   AxisStore[10].Axis[1..15].Pos13.Reached := FALSE;
   AxisStore[11].Axis[1..15].Pos13.Reached := FALSE;
   AxisStore[12].Axis[1..15].Pos13.Reached := FALSE;
   AxisStore[13].Axis[1..15].Pos13.Reached := FALSE;
   AxisStore[14].Axis[1..15].Pos13.Reached := FALSE;
   AxisStore[15].Axis[1..15].Pos13.Reached := FALSE;
   AxisStore[1].Axis[1..15].Pos14.Position := 0.0;
   AxisStore[2].Axis[1..15].Pos14.Position := 0.0;
   AxisStore[3].Axis[1..15].Pos14.Position := 0.0;
   AxisStore[4].Axis[1..15].Pos14.Position := 0.0;
   AxisStore[5].Axis[1..15].Pos14.Position := 0.0;
   AxisStore[6].Axis[1..15].Pos14.Position := 0.0;
   AxisStore[7].Axis[1..15].Pos14.Position := 0.0;
   AxisStore[8].Axis[1..15].Pos14.Position := 0.0;
   AxisStore[9].Axis[1..15].Pos14.Position := 0.0;
   AxisStore[10].Axis[1..15].Pos14.Position := 0.0;
   AxisStore[11].Axis[1..15].Pos14.Position := 0.0;
   AxisStore[12].Axis[1..15].Pos14.Position := 0.0;
   AxisStore[13].Axis[1..15].Pos14.Position := 0.0;
   AxisStore[14].Axis[1..15].Pos14.Position := 0.0;
   AxisStore[15].Axis[1..15].Pos14.Position := 0.0;
   AxisStore[1].Axis[1..15].Pos14.Speed := 0;
   AxisStore[2].Axis[1..15].Pos14.Speed := 0;
   AxisStore[3].Axis[1..15].Pos14.Speed := 0;
   AxisStore[4].Axis[1..15].Pos14.Speed := 0;
   AxisStore[5].Axis[1..15].Pos14.Speed := 0;
   AxisStore[6].Axis[1..15].Pos14.Speed := 0;
   AxisStore[7].Axis[1..15].Pos14.Speed := 0;
   AxisStore[8].Axis[1..15].Pos14.Speed := 0;
   AxisStore[9].Axis[1..15].Pos14.Speed := 0;
   AxisStore[10].Axis[1..15].Pos14.Speed := 0;
   AxisStore[11].Axis[1..15].Pos14.Speed := 0;
   AxisStore[12].Axis[1..15].Pos14.Speed := 0;
   AxisStore[13].Axis[1..15].Pos14.Speed := 0;
   AxisStore[14].Axis[1..15].Pos14.Speed := 0;
   AxisStore[15].Axis[1..15].Pos14.Speed := 0;
   AxisStore[1].Axis[1..15].Pos14.Reached := FALSE;
   AxisStore[2].Axis[1..15].Pos14.Reached := FALSE;
   AxisStore[3].Axis[1..15].Pos14.Reached := FALSE;
   AxisStore[4].Axis[1..15].Pos14.Reached := FALSE;
   AxisStore[5].Axis[1..15].Pos14.Reached := FALSE;
   AxisStore[6].Axis[1..15].Pos14.Reached := FALSE;
   AxisStore[7].Axis[1..15].Pos14.Reached := FALSE;
   AxisStore[8].Axis[1..15].Pos14.Reached := FALSE;
   AxisStore[9].Axis[1..15].Pos14.Reached := FALSE;
   AxisStore[10].Axis[1..15].Pos14.Reached := FALSE;
   AxisStore[11].Axis[1..15].Pos14.Reached := FALSE;
   AxisStore[12].Axis[1..15].Pos14.Reached := FALSE;
   AxisStore[13].Axis[1..15].Pos14.Reached := FALSE;
   AxisStore[14].Axis[1..15].Pos14.Reached := FALSE;
   AxisStore[15].Axis[1..15].Pos14.Reached := FALSE;
   AxisStore[1].Axis[1..15].Pos15.Position := 0.0;
   AxisStore[2].Axis[1..15].Pos15.Position := 0.0;
   AxisStore[3].Axis[1..15].Pos15.Position := 0.0;
   AxisStore[4].Axis[1..15].Pos15.Position := 0.0;
   AxisStore[5].Axis[1..15].Pos15.Position := 0.0;
   AxisStore[6].Axis[1..15].Pos15.Position := 0.0;
   AxisStore[7].Axis[1..15].Pos15.Position := 0.0;
   AxisStore[8].Axis[1..15].Pos15.Position := 0.0;
   AxisStore[9].Axis[1..15].Pos15.Position := 0.0;
   AxisStore[10].Axis[1..15].Pos15.Position := 0.0;
   AxisStore[11].Axis[1..15].Pos15.Position := 0.0;
   AxisStore[12].Axis[1..15].Pos15.Position := 0.0;
   AxisStore[13].Axis[1..15].Pos15.Position := 0.0;
   AxisStore[14].Axis[1..15].Pos15.Position := 0.0;
   AxisStore[15].Axis[1..15].Pos15.Position := 0.0;
   AxisStore[1].Axis[1..15].Pos15.Speed := 0;
   AxisStore[2].Axis[1..15].Pos15.Speed := 0;
   AxisStore[3].Axis[1..15].Pos15.Speed := 0;
   AxisStore[4].Axis[1..15].Pos15.Speed := 0;
   AxisStore[5].Axis[1..15].Pos15.Speed := 0;
   AxisStore[6].Axis[1..15].Pos15.Speed := 0;
   AxisStore[7].Axis[1..15].Pos15.Speed := 0;
   AxisStore[8].Axis[1..15].Pos15.Speed := 0;
   AxisStore[9].Axis[1..15].Pos15.Speed := 0;
   AxisStore[10].Axis[1..15].Pos15.Speed := 0;
   AxisStore[11].Axis[1..15].Pos15.Speed := 0;
   AxisStore[12].Axis[1..15].Pos15.Speed := 0;
   AxisStore[13].Axis[1..15].Pos15.Speed := 0;
   AxisStore[14].Axis[1..15].Pos15.Speed := 0;
   AxisStore[15].Axis[1..15].Pos15.Speed := 0;
   AxisStore[1].Axis[1..15].Pos15.Reached := FALSE;
   AxisStore[2].Axis[1..15].Pos15.Reached := FALSE;
   AxisStore[3].Axis[1..15].Pos15.Reached := FALSE;
   AxisStore[4].Axis[1..15].Pos15.Reached := FALSE;
   AxisStore[5].Axis[1..15].Pos15.Reached := FALSE;
   AxisStore[6].Axis[1..15].Pos15.Reached := FALSE;
   AxisStore[7].Axis[1..15].Pos15.Reached := FALSE;
   AxisStore[8].Axis[1..15].Pos15.Reached := FALSE;
   AxisStore[9].Axis[1..15].Pos15.Reached := FALSE;
   AxisStore[10].Axis[1..15].Pos15.Reached := FALSE;
   AxisStore[11].Axis[1..15].Pos15.Reached := FALSE;
   AxisStore[12].Axis[1..15].Pos15.Reached := FALSE;
   AxisStore[13].Axis[1..15].Pos15.Reached := FALSE;
   AxisStore[14].Axis[1..15].Pos15.Reached := FALSE;
   AxisStore[15].Axis[1..15].Pos15.Reached := FALSE;
   AxisStore[1].Axis[1..15].Pos16.Position := 0.0;
   AxisStore[2].Axis[1..15].Pos16.Position := 0.0;
   AxisStore[3].Axis[1..15].Pos16.Position := 0.0;
   AxisStore[4].Axis[1..15].Pos16.Position := 0.0;
   AxisStore[5].Axis[1..15].Pos16.Position := 0.0;
   AxisStore[6].Axis[1..15].Pos16.Position := 0.0;
   AxisStore[7].Axis[1..15].Pos16.Position := 0.0;
   AxisStore[8].Axis[1..15].Pos16.Position := 0.0;
   AxisStore[9].Axis[1..15].Pos16.Position := 0.0;
   AxisStore[10].Axis[1..15].Pos16.Position := 0.0;
   AxisStore[11].Axis[1..15].Pos16.Position := 0.0;
   AxisStore[12].Axis[1..15].Pos16.Position := 0.0;
   AxisStore[13].Axis[1..15].Pos16.Position := 0.0;
   AxisStore[14].Axis[1..15].Pos16.Position := 0.0;
   AxisStore[15].Axis[1..15].Pos16.Position := 0.0;
   AxisStore[1].Axis[1..15].Pos16.Speed := 0;
   AxisStore[2].Axis[1..15].Pos16.Speed := 0;
   AxisStore[3].Axis[1..15].Pos16.Speed := 0;
   AxisStore[4].Axis[1..15].Pos16.Speed := 0;
   AxisStore[5].Axis[1..15].Pos16.Speed := 0;
   AxisStore[6].Axis[1..15].Pos16.Speed := 0;
   AxisStore[7].Axis[1..15].Pos16.Speed := 0;
   AxisStore[8].Axis[1..15].Pos16.Speed := 0;
   AxisStore[9].Axis[1..15].Pos16.Speed := 0;
   AxisStore[10].Axis[1..15].Pos16.Speed := 0;
   AxisStore[11].Axis[1..15].Pos16.Speed := 0;
   AxisStore[12].Axis[1..15].Pos16.Speed := 0;
   AxisStore[13].Axis[1..15].Pos16.Speed := 0;
   AxisStore[14].Axis[1..15].Pos16.Speed := 0;
   AxisStore[15].Axis[1..15].Pos16.Speed := 0;
   AxisStore[1].Axis[1..15].Pos16.Reached := FALSE;
   AxisStore[2].Axis[1..15].Pos16.Reached := FALSE;
   AxisStore[3].Axis[1..15].Pos16.Reached := FALSE;
   AxisStore[4].Axis[1..15].Pos16.Reached := FALSE;
   AxisStore[5].Axis[1..15].Pos16.Reached := FALSE;
   AxisStore[6].Axis[1..15].Pos16.Reached := FALSE;
   AxisStore[7].Axis[1..15].Pos16.Reached := FALSE;
   AxisStore[8].Axis[1..15].Pos16.Reached := FALSE;
   AxisStore[9].Axis[1..15].Pos16.Reached := FALSE;
   AxisStore[10].Axis[1..15].Pos16.Reached := FALSE;
   AxisStore[11].Axis[1..15].Pos16.Reached := FALSE;
   AxisStore[12].Axis[1..15].Pos16.Reached := FALSE;
   AxisStore[13].Axis[1..15].Pos16.Reached := FALSE;
   AxisStore[14].Axis[1..15].Pos16.Reached := FALSE;
   AxisStore[15].Axis[1..15].Pos16.Reached := FALSE;
   AxisStore[1].Axis[1..15].Pos17.Position := 0.0;
   AxisStore[2].Axis[1..15].Pos17.Position := 0.0;
   AxisStore[3].Axis[1..15].Pos17.Position := 0.0;
   AxisStore[4].Axis[1..15].Pos17.Position := 0.0;
   AxisStore[5].Axis[1..15].Pos17.Position := 0.0;
   AxisStore[6].Axis[1..15].Pos17.Position := 0.0;
   AxisStore[7].Axis[1..15].Pos17.Position := 0.0;
   AxisStore[8].Axis[1..15].Pos17.Position := 0.0;
   AxisStore[9].Axis[1..15].Pos17.Position := 0.0;
   AxisStore[10].Axis[1..15].Pos17.Position := 0.0;
   AxisStore[11].Axis[1..15].Pos17.Position := 0.0;
   AxisStore[12].Axis[1..15].Pos17.Position := 0.0;
   AxisStore[13].Axis[1..15].Pos17.Position := 0.0;
   AxisStore[14].Axis[1..15].Pos17.Position := 0.0;
   AxisStore[15].Axis[1..15].Pos17.Position := 0.0;
   AxisStore[1].Axis[1..15].Pos17.Speed := 0;
   AxisStore[2].Axis[1..15].Pos17.Speed := 0;
   AxisStore[3].Axis[1..15].Pos17.Speed := 0;
   AxisStore[4].Axis[1..15].Pos17.Speed := 0;
   AxisStore[5].Axis[1..15].Pos17.Speed := 0;
   AxisStore[6].Axis[1..15].Pos17.Speed := 0;
   AxisStore[7].Axis[1..15].Pos17.Speed := 0;
   AxisStore[8].Axis[1..15].Pos17.Speed := 0;
   AxisStore[9].Axis[1..15].Pos17.Speed := 0;
   AxisStore[10].Axis[1..15].Pos17.Speed := 0;
   AxisStore[11].Axis[1..15].Pos17.Speed := 0;
   AxisStore[12].Axis[1..15].Pos17.Speed := 0;
   AxisStore[13].Axis[1..15].Pos17.Speed := 0;
   AxisStore[14].Axis[1..15].Pos17.Speed := 0;
   AxisStore[15].Axis[1..15].Pos17.Speed := 0;
   AxisStore[1].Axis[1..15].Pos17.Reached := FALSE;
   AxisStore[2].Axis[1..15].Pos17.Reached := FALSE;
   AxisStore[3].Axis[1..15].Pos17.Reached := FALSE;
   AxisStore[4].Axis[1..15].Pos17.Reached := FALSE;
   AxisStore[5].Axis[1..15].Pos17.Reached := FALSE;
   AxisStore[6].Axis[1..15].Pos17.Reached := FALSE;
   AxisStore[7].Axis[1..15].Pos17.Reached := FALSE;
   AxisStore[8].Axis[1..15].Pos17.Reached := FALSE;
   AxisStore[9].Axis[1..15].Pos17.Reached := FALSE;
   AxisStore[10].Axis[1..15].Pos17.Reached := FALSE;
   AxisStore[11].Axis[1..15].Pos17.Reached := FALSE;
   AxisStore[12].Axis[1..15].Pos17.Reached := FALSE;
   AxisStore[13].Axis[1..15].Pos17.Reached := FALSE;
   AxisStore[14].Axis[1..15].Pos17.Reached := FALSE;
   AxisStore[15].Axis[1..15].Pos17.Reached := FALSE;
   AxisStore[1].Axis[1..15].Pos18.Position := 0.0;
   AxisStore[2].Axis[1..15].Pos18.Position := 0.0;
   AxisStore[3].Axis[1..15].Pos18.Position := 0.0;
   AxisStore[4].Axis[1..15].Pos18.Position := 0.0;
   AxisStore[5].Axis[1..15].Pos18.Position := 0.0;
   AxisStore[6].Axis[1..15].Pos18.Position := 0.0;
   AxisStore[7].Axis[1..15].Pos18.Position := 0.0;
   AxisStore[8].Axis[1..15].Pos18.Position := 0.0;
   AxisStore[9].Axis[1..15].Pos18.Position := 0.0;
   AxisStore[10].Axis[1..15].Pos18.Position := 0.0;
   AxisStore[11].Axis[1..15].Pos18.Position := 0.0;
   AxisStore[12].Axis[1..15].Pos18.Position := 0.0;
   AxisStore[13].Axis[1..15].Pos18.Position := 0.0;
   AxisStore[14].Axis[1..15].Pos18.Position := 0.0;
   AxisStore[15].Axis[1..15].Pos18.Position := 0.0;
   AxisStore[1].Axis[1..15].Pos18.Speed := 0;
   AxisStore[2].Axis[1..15].Pos18.Speed := 0;
   AxisStore[3].Axis[1..15].Pos18.Speed := 0;
   AxisStore[4].Axis[1..15].Pos18.Speed := 0;
   AxisStore[5].Axis[1..15].Pos18.Speed := 0;
   AxisStore[6].Axis[1..15].Pos18.Speed := 0;
   AxisStore[7].Axis[1..15].Pos18.Speed := 0;
   AxisStore[8].Axis[1..15].Pos18.Speed := 0;
   AxisStore[9].Axis[1..15].Pos18.Speed := 0;
   AxisStore[10].Axis[1..15].Pos18.Speed := 0;
   AxisStore[11].Axis[1..15].Pos18.Speed := 0;
   AxisStore[12].Axis[1..15].Pos18.Speed := 0;
   AxisStore[13].Axis[1..15].Pos18.Speed := 0;
   AxisStore[14].Axis[1..15].Pos18.Speed := 0;
   AxisStore[15].Axis[1..15].Pos18.Speed := 0;
   AxisStore[1].Axis[1..15].Pos18.Reached := FALSE;
   AxisStore[2].Axis[1..15].Pos18.Reached := FALSE;
   AxisStore[3].Axis[1..15].Pos18.Reached := FALSE;
   AxisStore[4].Axis[1..15].Pos18.Reached := FALSE;
   AxisStore[5].Axis[1..15].Pos18.Reached := FALSE;
   AxisStore[6].Axis[1..15].Pos18.Reached := FALSE;
   AxisStore[7].Axis[1..15].Pos18.Reached := FALSE;
   AxisStore[8].Axis[1..15].Pos18.Reached := FALSE;
   AxisStore[9].Axis[1..15].Pos18.Reached := FALSE;
   AxisStore[10].Axis[1..15].Pos18.Reached := FALSE;
   AxisStore[11].Axis[1..15].Pos18.Reached := FALSE;
   AxisStore[12].Axis[1..15].Pos18.Reached := FALSE;
   AxisStore[13].Axis[1..15].Pos18.Reached := FALSE;
   AxisStore[14].Axis[1..15].Pos18.Reached := FALSE;
   AxisStore[15].Axis[1..15].Pos18.Reached := FALSE;
   AxisStore[1].Axis[1..15].Pos19.Position := 0.0;
   AxisStore[2].Axis[1..15].Pos19.Position := 0.0;
   AxisStore[3].Axis[1..15].Pos19.Position := 0.0;
   AxisStore[4].Axis[1..15].Pos19.Position := 0.0;
   AxisStore[5].Axis[1..15].Pos19.Position := 0.0;
   AxisStore[6].Axis[1..15].Pos19.Position := 0.0;
   AxisStore[7].Axis[1..15].Pos19.Position := 0.0;
   AxisStore[8].Axis[1..15].Pos19.Position := 0.0;
   AxisStore[9].Axis[1..15].Pos19.Position := 0.0;
   AxisStore[10].Axis[1..15].Pos19.Position := 0.0;
   AxisStore[11].Axis[1..15].Pos19.Position := 0.0;
   AxisStore[12].Axis[1..15].Pos19.Position := 0.0;
   AxisStore[13].Axis[1..15].Pos19.Position := 0.0;
   AxisStore[14].Axis[1..15].Pos19.Position := 0.0;
   AxisStore[15].Axis[1..15].Pos19.Position := 0.0;
   AxisStore[1].Axis[1..15].Pos19.Speed := 0;
   AxisStore[2].Axis[1..15].Pos19.Speed := 0;
   AxisStore[3].Axis[1..15].Pos19.Speed := 0;
   AxisStore[4].Axis[1..15].Pos19.Speed := 0;
   AxisStore[5].Axis[1..15].Pos19.Speed := 0;
   AxisStore[6].Axis[1..15].Pos19.Speed := 0;
   AxisStore[7].Axis[1..15].Pos19.Speed := 0;
   AxisStore[8].Axis[1..15].Pos19.Speed := 0;
   AxisStore[9].Axis[1..15].Pos19.Speed := 0;
   AxisStore[10].Axis[1..15].Pos19.Speed := 0;
   AxisStore[11].Axis[1..15].Pos19.Speed := 0;
   AxisStore[12].Axis[1..15].Pos19.Speed := 0;
   AxisStore[13].Axis[1..15].Pos19.Speed := 0;
   AxisStore[14].Axis[1..15].Pos19.Speed := 0;
   AxisStore[15].Axis[1..15].Pos19.Speed := 0;
   AxisStore[1].Axis[1..15].Pos19.Reached := FALSE;
   AxisStore[2].Axis[1..15].Pos19.Reached := FALSE;
   AxisStore[3].Axis[1..15].Pos19.Reached := FALSE;
   AxisStore[4].Axis[1..15].Pos19.Reached := FALSE;
   AxisStore[5].Axis[1..15].Pos19.Reached := FALSE;
   AxisStore[6].Axis[1..15].Pos19.Reached := FALSE;
   AxisStore[7].Axis[1..15].Pos19.Reached := FALSE;
   AxisStore[8].Axis[1..15].Pos19.Reached := FALSE;
   AxisStore[9].Axis[1..15].Pos19.Reached := FALSE;
   AxisStore[10].Axis[1..15].Pos19.Reached := FALSE;
   AxisStore[11].Axis[1..15].Pos19.Reached := FALSE;
   AxisStore[12].Axis[1..15].Pos19.Reached := FALSE;
   AxisStore[13].Axis[1..15].Pos19.Reached := FALSE;
   AxisStore[14].Axis[1..15].Pos19.Reached := FALSE;
   AxisStore[15].Axis[1..15].Pos19.Reached := FALSE;
   AxisStore[1].Axis[1..15].Pos20.Position := 0.0;
   AxisStore[2].Axis[1..15].Pos20.Position := 0.0;
   AxisStore[3].Axis[1..15].Pos20.Position := 0.0;
   AxisStore[4].Axis[1..15].Pos20.Position := 0.0;
   AxisStore[5].Axis[1..15].Pos20.Position := 0.0;
   AxisStore[6].Axis[1..15].Pos20.Position := 0.0;
   AxisStore[7].Axis[1..15].Pos20.Position := 0.0;
   AxisStore[8].Axis[1..15].Pos20.Position := 0.0;
   AxisStore[9].Axis[1..15].Pos20.Position := 0.0;
   AxisStore[10].Axis[1..15].Pos20.Position := 0.0;
   AxisStore[11].Axis[1..15].Pos20.Position := 0.0;
   AxisStore[12].Axis[1..15].Pos20.Position := 0.0;
   AxisStore[13].Axis[1..15].Pos20.Position := 0.0;
   AxisStore[14].Axis[1..15].Pos20.Position := 0.0;
   AxisStore[15].Axis[1..15].Pos20.Position := 0.0;
   AxisStore[1].Axis[1..15].Pos20.Speed := 0;
   AxisStore[2].Axis[1..15].Pos20.Speed := 0;
   AxisStore[3].Axis[1..15].Pos20.Speed := 0;
   AxisStore[4].Axis[1..15].Pos20.Speed := 0;
   AxisStore[5].Axis[1..15].Pos20.Speed := 0;
   AxisStore[6].Axis[1..15].Pos20.Speed := 0;
   AxisStore[7].Axis[1..15].Pos20.Speed := 0;
   AxisStore[8].Axis[1..15].Pos20.Speed := 0;
   AxisStore[9].Axis[1..15].Pos20.Speed := 0;
   AxisStore[10].Axis[1..15].Pos20.Speed := 0;
   AxisStore[11].Axis[1..15].Pos20.Speed := 0;
   AxisStore[12].Axis[1..15].Pos20.Speed := 0;
   AxisStore[13].Axis[1..15].Pos20.Speed := 0;
   AxisStore[14].Axis[1..15].Pos20.Speed := 0;
   AxisStore[15].Axis[1..15].Pos20.Speed := 0;
   AxisStore[1].Axis[1..15].Pos20.Reached := FALSE;
   AxisStore[2].Axis[1..15].Pos20.Reached := FALSE;
   AxisStore[3].Axis[1..15].Pos20.Reached := FALSE;
   AxisStore[4].Axis[1..15].Pos20.Reached := FALSE;
   AxisStore[5].Axis[1..15].Pos20.Reached := FALSE;
   AxisStore[6].Axis[1..15].Pos20.Reached := FALSE;
   AxisStore[7].Axis[1..15].Pos20.Reached := FALSE;
   AxisStore[8].Axis[1..15].Pos20.Reached := FALSE;
   AxisStore[9].Axis[1..15].Pos20.Reached := FALSE;
   AxisStore[10].Axis[1..15].Pos20.Reached := FALSE;
   AxisStore[11].Axis[1..15].Pos20.Reached := FALSE;
   AxisStore[12].Axis[1..15].Pos20.Reached := FALSE;
   AxisStore[13].Axis[1..15].Pos20.Reached := FALSE;
   AxisStore[14].Axis[1..15].Pos20.Reached := FALSE;
   AxisStore[15].Axis[1..15].Pos20.Reached := FALSE;
   AxisStore[1].Axis[1..15].Pos21.Position := 0.0;
   AxisStore[2].Axis[1..15].Pos21.Position := 0.0;
   AxisStore[3].Axis[1..15].Pos21.Position := 0.0;
   AxisStore[4].Axis[1..15].Pos21.Position := 0.0;
   AxisStore[5].Axis[1..15].Pos21.Position := 0.0;
   AxisStore[6].Axis[1..15].Pos21.Position := 0.0;
   AxisStore[7].Axis[1..15].Pos21.Position := 0.0;
   AxisStore[8].Axis[1..15].Pos21.Position := 0.0;
   AxisStore[9].Axis[1..15].Pos21.Position := 0.0;
   AxisStore[10].Axis[1..15].Pos21.Position := 0.0;
   AxisStore[11].Axis[1..15].Pos21.Position := 0.0;
   AxisStore[12].Axis[1..15].Pos21.Position := 0.0;
   AxisStore[13].Axis[1..15].Pos21.Position := 0.0;
   AxisStore[14].Axis[1..15].Pos21.Position := 0.0;
   AxisStore[15].Axis[1..15].Pos21.Position := 0.0;
   AxisStore[1].Axis[1..15].Pos21.Speed := 0;
   AxisStore[2].Axis[1..15].Pos21.Speed := 0;
   AxisStore[3].Axis[1..15].Pos21.Speed := 0;
   AxisStore[4].Axis[1..15].Pos21.Speed := 0;
   AxisStore[5].Axis[1..15].Pos21.Speed := 0;
   AxisStore[6].Axis[1..15].Pos21.Speed := 0;
   AxisStore[7].Axis[1..15].Pos21.Speed := 0;
   AxisStore[8].Axis[1..15].Pos21.Speed := 0;
   AxisStore[9].Axis[1..15].Pos21.Speed := 0;
   AxisStore[10].Axis[1..15].Pos21.Speed := 0;
   AxisStore[11].Axis[1..15].Pos21.Speed := 0;
   AxisStore[12].Axis[1..15].Pos21.Speed := 0;
   AxisStore[13].Axis[1..15].Pos21.Speed := 0;
   AxisStore[14].Axis[1..15].Pos21.Speed := 0;
   AxisStore[15].Axis[1..15].Pos21.Speed := 0;
   AxisStore[1].Axis[1..15].Pos21.Reached := FALSE;
   AxisStore[2].Axis[1..15].Pos21.Reached := FALSE;
   AxisStore[3].Axis[1..15].Pos21.Reached := FALSE;
   AxisStore[4].Axis[1..15].Pos21.Reached := FALSE;
   AxisStore[5].Axis[1..15].Pos21.Reached := FALSE;
   AxisStore[6].Axis[1..15].Pos21.Reached := FALSE;
   AxisStore[7].Axis[1..15].Pos21.Reached := FALSE;
   AxisStore[8].Axis[1..15].Pos21.Reached := FALSE;
   AxisStore[9].Axis[1..15].Pos21.Reached := FALSE;
   AxisStore[10].Axis[1..15].Pos21.Reached := FALSE;
   AxisStore[11].Axis[1..15].Pos21.Reached := FALSE;
   AxisStore[12].Axis[1..15].Pos21.Reached := FALSE;
   AxisStore[13].Axis[1..15].Pos21.Reached := FALSE;
   AxisStore[14].Axis[1..15].Pos21.Reached := FALSE;
   AxisStore[15].Axis[1..15].Pos21.Reached := FALSE;
   AxisStore[1].Axis[1..15].Pos22.Position := 0.0;
   AxisStore[2].Axis[1..15].Pos22.Position := 0.0;
   AxisStore[3].Axis[1..15].Pos22.Position := 0.0;
   AxisStore[4].Axis[1..15].Pos22.Position := 0.0;
   AxisStore[5].Axis[1..15].Pos22.Position := 0.0;
   AxisStore[6].Axis[1..15].Pos22.Position := 0.0;
   AxisStore[7].Axis[1..15].Pos22.Position := 0.0;
   AxisStore[8].Axis[1..15].Pos22.Position := 0.0;
   AxisStore[9].Axis[1..15].Pos22.Position := 0.0;
   AxisStore[10].Axis[1..15].Pos22.Position := 0.0;
   AxisStore[11].Axis[1..15].Pos22.Position := 0.0;
   AxisStore[12].Axis[1..15].Pos22.Position := 0.0;
   AxisStore[13].Axis[1..15].Pos22.Position := 0.0;
   AxisStore[14].Axis[1..15].Pos22.Position := 0.0;
   AxisStore[15].Axis[1..15].Pos22.Position := 0.0;
   AxisStore[1].Axis[1..15].Pos22.Speed := 0;
   AxisStore[2].Axis[1..15].Pos22.Speed := 0;
   AxisStore[3].Axis[1..15].Pos22.Speed := 0;
   AxisStore[4].Axis[1..15].Pos22.Speed := 0;
   AxisStore[5].Axis[1..15].Pos22.Speed := 0;
   AxisStore[6].Axis[1..15].Pos22.Speed := 0;
   AxisStore[7].Axis[1..15].Pos22.Speed := 0;
   AxisStore[8].Axis[1..15].Pos22.Speed := 0;
   AxisStore[9].Axis[1..15].Pos22.Speed := 0;
   AxisStore[10].Axis[1..15].Pos22.Speed := 0;
   AxisStore[11].Axis[1..15].Pos22.Speed := 0;
   AxisStore[12].Axis[1..15].Pos22.Speed := 0;
   AxisStore[13].Axis[1..15].Pos22.Speed := 0;
   AxisStore[14].Axis[1..15].Pos22.Speed := 0;
   AxisStore[15].Axis[1..15].Pos22.Speed := 0;
   AxisStore[1].Axis[1..15].Pos22.Reached := FALSE;
   AxisStore[2].Axis[1..15].Pos22.Reached := FALSE;
   AxisStore[3].Axis[1..15].Pos22.Reached := FALSE;
   AxisStore[4].Axis[1..15].Pos22.Reached := FALSE;
   AxisStore[5].Axis[1..15].Pos22.Reached := FALSE;
   AxisStore[6].Axis[1..15].Pos22.Reached := FALSE;
   AxisStore[7].Axis[1..15].Pos22.Reached := FALSE;
   AxisStore[8].Axis[1..15].Pos22.Reached := FALSE;
   AxisStore[9].Axis[1..15].Pos22.Reached := FALSE;
   AxisStore[10].Axis[1..15].Pos22.Reached := FALSE;
   AxisStore[11].Axis[1..15].Pos22.Reached := FALSE;
   AxisStore[12].Axis[1..15].Pos22.Reached := FALSE;
   AxisStore[13].Axis[1..15].Pos22.Reached := FALSE;
   AxisStore[14].Axis[1..15].Pos22.Reached := FALSE;
   AxisStore[15].Axis[1..15].Pos22.Reached := FALSE;
   AxisStore[1].Axis[1..15].Pos23.Position := 0.0;
   AxisStore[2].Axis[1..15].Pos23.Position := 0.0;
   AxisStore[3].Axis[1..15].Pos23.Position := 0.0;
   AxisStore[4].Axis[1..15].Pos23.Position := 0.0;
   AxisStore[5].Axis[1..15].Pos23.Position := 0.0;
   AxisStore[6].Axis[1..15].Pos23.Position := 0.0;
   AxisStore[7].Axis[1..15].Pos23.Position := 0.0;
   AxisStore[8].Axis[1..15].Pos23.Position := 0.0;
   AxisStore[9].Axis[1..15].Pos23.Position := 0.0;
   AxisStore[10].Axis[1..15].Pos23.Position := 0.0;
   AxisStore[11].Axis[1..15].Pos23.Position := 0.0;
   AxisStore[12].Axis[1..15].Pos23.Position := 0.0;
   AxisStore[13].Axis[1..15].Pos23.Position := 0.0;
   AxisStore[14].Axis[1..15].Pos23.Position := 0.0;
   AxisStore[15].Axis[1..15].Pos23.Position := 0.0;
   AxisStore[1].Axis[1..15].Pos23.Speed := 0;
   AxisStore[2].Axis[1..15].Pos23.Speed := 0;
   AxisStore[3].Axis[1..15].Pos23.Speed := 0;
   AxisStore[4].Axis[1..15].Pos23.Speed := 0;
   AxisStore[5].Axis[1..15].Pos23.Speed := 0;
   AxisStore[6].Axis[1..15].Pos23.Speed := 0;
   AxisStore[7].Axis[1..15].Pos23.Speed := 0;
   AxisStore[8].Axis[1..15].Pos23.Speed := 0;
   AxisStore[9].Axis[1..15].Pos23.Speed := 0;
   AxisStore[10].Axis[1..15].Pos23.Speed := 0;
   AxisStore[11].Axis[1..15].Pos23.Speed := 0;
   AxisStore[12].Axis[1..15].Pos23.Speed := 0;
   AxisStore[13].Axis[1..15].Pos23.Speed := 0;
   AxisStore[14].Axis[1..15].Pos23.Speed := 0;
   AxisStore[15].Axis[1..15].Pos23.Speed := 0;
   AxisStore[1].Axis[1..15].Pos23.Reached := FALSE;
   AxisStore[2].Axis[1..15].Pos23.Reached := FALSE;
   AxisStore[3].Axis[1..15].Pos23.Reached := FALSE;
   AxisStore[4].Axis[1..15].Pos23.Reached := FALSE;
   AxisStore[5].Axis[1..15].Pos23.Reached := FALSE;
   AxisStore[6].Axis[1..15].Pos23.Reached := FALSE;
   AxisStore[7].Axis[1..15].Pos23.Reached := FALSE;
   AxisStore[8].Axis[1..15].Pos23.Reached := FALSE;
   AxisStore[9].Axis[1..15].Pos23.Reached := FALSE;
   AxisStore[10].Axis[1..15].Pos23.Reached := FALSE;
   AxisStore[11].Axis[1..15].Pos23.Reached := FALSE;
   AxisStore[12].Axis[1..15].Pos23.Reached := FALSE;
   AxisStore[13].Axis[1..15].Pos23.Reached := FALSE;
   AxisStore[14].Axis[1..15].Pos23.Reached := FALSE;
   AxisStore[15].Axis[1..15].Pos23.Reached := FALSE;
   AxisStore[1].Axis[1..15].Pos24.Position := 0.0;
   AxisStore[2].Axis[1..15].Pos24.Position := 0.0;
   AxisStore[3].Axis[1..15].Pos24.Position := 0.0;
   AxisStore[4].Axis[1..15].Pos24.Position := 0.0;
   AxisStore[5].Axis[1..15].Pos24.Position := 0.0;
   AxisStore[6].Axis[1..15].Pos24.Position := 0.0;
   AxisStore[7].Axis[1..15].Pos24.Position := 0.0;
   AxisStore[8].Axis[1..15].Pos24.Position := 0.0;
   AxisStore[9].Axis[1..15].Pos24.Position := 0.0;
   AxisStore[10].Axis[1..15].Pos24.Position := 0.0;
   AxisStore[11].Axis[1..15].Pos24.Position := 0.0;
   AxisStore[12].Axis[1..15].Pos24.Position := 0.0;
   AxisStore[13].Axis[1..15].Pos24.Position := 0.0;
   AxisStore[14].Axis[1..15].Pos24.Position := 0.0;
   AxisStore[15].Axis[1..15].Pos24.Position := 0.0;
   AxisStore[1].Axis[1..15].Pos24.Speed := 0;
   AxisStore[2].Axis[1..15].Pos24.Speed := 0;
   AxisStore[3].Axis[1..15].Pos24.Speed := 0;
   AxisStore[4].Axis[1..15].Pos24.Speed := 0;
   AxisStore[5].Axis[1..15].Pos24.Speed := 0;
   AxisStore[6].Axis[1..15].Pos24.Speed := 0;
   AxisStore[7].Axis[1..15].Pos24.Speed := 0;
   AxisStore[8].Axis[1..15].Pos24.Speed := 0;
   AxisStore[9].Axis[1..15].Pos24.Speed := 0;
   AxisStore[10].Axis[1..15].Pos24.Speed := 0;
   AxisStore[11].Axis[1..15].Pos24.Speed := 0;
   AxisStore[12].Axis[1..15].Pos24.Speed := 0;
   AxisStore[13].Axis[1..15].Pos24.Speed := 0;
   AxisStore[14].Axis[1..15].Pos24.Speed := 0;
   AxisStore[15].Axis[1..15].Pos24.Speed := 0;
   AxisStore[1].Axis[1..15].Pos24.Reached := FALSE;
   AxisStore[2].Axis[1..15].Pos24.Reached := FALSE;
   AxisStore[3].Axis[1..15].Pos24.Reached := FALSE;
   AxisStore[4].Axis[1..15].Pos24.Reached := FALSE;
   AxisStore[5].Axis[1..15].Pos24.Reached := FALSE;
   AxisStore[6].Axis[1..15].Pos24.Reached := FALSE;
   AxisStore[7].Axis[1..15].Pos24.Reached := FALSE;
   AxisStore[8].Axis[1..15].Pos24.Reached := FALSE;
   AxisStore[9].Axis[1..15].Pos24.Reached := FALSE;
   AxisStore[10].Axis[1..15].Pos24.Reached := FALSE;
   AxisStore[11].Axis[1..15].Pos24.Reached := FALSE;
   AxisStore[12].Axis[1..15].Pos24.Reached := FALSE;
   AxisStore[13].Axis[1..15].Pos24.Reached := FALSE;
   AxisStore[14].Axis[1..15].Pos24.Reached := FALSE;
   AxisStore[15].Axis[1..15].Pos24.Reached := FALSE;
   AxisStore[1].Axis[1..15].Pos25.Position := 0.0;
   AxisStore[2].Axis[1..15].Pos25.Position := 0.0;
   AxisStore[3].Axis[1..15].Pos25.Position := 0.0;
   AxisStore[4].Axis[1..15].Pos25.Position := 0.0;
   AxisStore[5].Axis[1..15].Pos25.Position := 0.0;
   AxisStore[6].Axis[1..15].Pos25.Position := 0.0;
   AxisStore[7].Axis[1..15].Pos25.Position := 0.0;
   AxisStore[8].Axis[1..15].Pos25.Position := 0.0;
   AxisStore[9].Axis[1..15].Pos25.Position := 0.0;
   AxisStore[10].Axis[1..15].Pos25.Position := 0.0;
   AxisStore[11].Axis[1..15].Pos25.Position := 0.0;
   AxisStore[12].Axis[1..15].Pos25.Position := 0.0;
   AxisStore[13].Axis[1..15].Pos25.Position := 0.0;
   AxisStore[14].Axis[1..15].Pos25.Position := 0.0;
   AxisStore[15].Axis[1..15].Pos25.Position := 0.0;
   AxisStore[1].Axis[1..15].Pos25.Speed := 0;
   AxisStore[2].Axis[1..15].Pos25.Speed := 0;
   AxisStore[3].Axis[1..15].Pos25.Speed := 0;
   AxisStore[4].Axis[1..15].Pos25.Speed := 0;
   AxisStore[5].Axis[1..15].Pos25.Speed := 0;
   AxisStore[6].Axis[1..15].Pos25.Speed := 0;
   AxisStore[7].Axis[1..15].Pos25.Speed := 0;
   AxisStore[8].Axis[1..15].Pos25.Speed := 0;
   AxisStore[9].Axis[1..15].Pos25.Speed := 0;
   AxisStore[10].Axis[1..15].Pos25.Speed := 0;
   AxisStore[11].Axis[1..15].Pos25.Speed := 0;
   AxisStore[12].Axis[1..15].Pos25.Speed := 0;
   AxisStore[13].Axis[1..15].Pos25.Speed := 0;
   AxisStore[14].Axis[1..15].Pos25.Speed := 0;
   AxisStore[15].Axis[1..15].Pos25.Speed := 0;
   AxisStore[1].Axis[1..15].Pos25.Reached := FALSE;
   AxisStore[2].Axis[1..15].Pos25.Reached := FALSE;
   AxisStore[3].Axis[1..15].Pos25.Reached := FALSE;
   AxisStore[4].Axis[1..15].Pos25.Reached := FALSE;
   AxisStore[5].Axis[1..15].Pos25.Reached := FALSE;
   AxisStore[6].Axis[1..15].Pos25.Reached := FALSE;
   AxisStore[7].Axis[1..15].Pos25.Reached := FALSE;
   AxisStore[8].Axis[1..15].Pos25.Reached := FALSE;
   AxisStore[9].Axis[1..15].Pos25.Reached := FALSE;
   AxisStore[10].Axis[1..15].Pos25.Reached := FALSE;
   AxisStore[11].Axis[1..15].Pos25.Reached := FALSE;
   AxisStore[12].Axis[1..15].Pos25.Reached := FALSE;
   AxisStore[13].Axis[1..15].Pos25.Reached := FALSE;
   AxisStore[14].Axis[1..15].Pos25.Reached := FALSE;
   AxisStore[15].Axis[1..15].Pos25.Reached := FALSE;
   AxisStore[1].Axis[1..15].Pos26.Position := 0.0;
   AxisStore[2].Axis[1..15].Pos26.Position := 0.0;
   AxisStore[3].Axis[1..15].Pos26.Position := 0.0;
   AxisStore[4].Axis[1..15].Pos26.Position := 0.0;
   AxisStore[5].Axis[1..15].Pos26.Position := 0.0;
   AxisStore[6].Axis[1..15].Pos26.Position := 0.0;
   AxisStore[7].Axis[1..15].Pos26.Position := 0.0;
   AxisStore[8].Axis[1..15].Pos26.Position := 0.0;
   AxisStore[9].Axis[1..15].Pos26.Position := 0.0;
   AxisStore[10].Axis[1..15].Pos26.Position := 0.0;
   AxisStore[11].Axis[1..15].Pos26.Position := 0.0;
   AxisStore[12].Axis[1..15].Pos26.Position := 0.0;
   AxisStore[13].Axis[1..15].Pos26.Position := 0.0;
   AxisStore[14].Axis[1..15].Pos26.Position := 0.0;
   AxisStore[15].Axis[1..15].Pos26.Position := 0.0;
   AxisStore[1].Axis[1..15].Pos26.Speed := 0;
   AxisStore[2].Axis[1..15].Pos26.Speed := 0;
   AxisStore[3].Axis[1..15].Pos26.Speed := 0;
   AxisStore[4].Axis[1..15].Pos26.Speed := 0;
   AxisStore[5].Axis[1..15].Pos26.Speed := 0;
   AxisStore[6].Axis[1..15].Pos26.Speed := 0;
   AxisStore[7].Axis[1..15].Pos26.Speed := 0;
   AxisStore[8].Axis[1..15].Pos26.Speed := 0;
   AxisStore[9].Axis[1..15].Pos26.Speed := 0;
   AxisStore[10].Axis[1..15].Pos26.Speed := 0;
   AxisStore[11].Axis[1..15].Pos26.Speed := 0;
   AxisStore[12].Axis[1..15].Pos26.Speed := 0;
   AxisStore[13].Axis[1..15].Pos26.Speed := 0;
   AxisStore[14].Axis[1..15].Pos26.Speed := 0;
   AxisStore[15].Axis[1..15].Pos26.Speed := 0;
   AxisStore[1].Axis[1..15].Pos26.Reached := FALSE;
   AxisStore[2].Axis[1..15].Pos26.Reached := FALSE;
   AxisStore[3].Axis[1..15].Pos26.Reached := FALSE;
   AxisStore[4].Axis[1..15].Pos26.Reached := FALSE;
